(* CODESYS project CtaAppSperrAntrieb_2.0.0.0.library
   Description: Sperr- Antriebs Library der CTA
   Version: 2.0.0.0
   Title: CtaAppSperrAntrieb
   Author: SIS
   DocFormat: reStructuredText
   Placeholder: CtaAppSperrAntrieb
   LanguageModelAttribute: qualified-access-only
   CompiledLibraryCompatibilityVersion: CODESYS V3.5 SP16 Patch 3
   Company: CTA
   DefaultNamespace: CtaAppSperrAntrieb

Project tree, tasks and I/O mapping:
  libraries: Standard, 3.5.18.0 (System); CtaAppBasic, 1.0.0.0 (CTA); CtaAppBmk, 2.0.0.0 (CTA); CtaAppReport, 2.0.0.0 (CTA); CtaSysConfig, 2.0.0.0 (CTA); VisuSymbols, 4.5.0.0 (System); VisuDialogs, 3.5.16.20 (System); CtaSysMotor, 1.0.0.0 (CTA); CtaVisHelp, 1.0.0.0 (CTA); CtaVisSymbols, 2.0.0.0 (CTA); CtaSysIO, 2.0.0.0 (CTA); CtaAppInfluxLog, 1.0.0.1 (CTA); CtaAppModbusSpezifikation, 1.0.0.1 (CTA); CtaVisApps, 1.0.0.0 (CTA); CtaVisUser, 1.0.0.0 (CTA)
  40 Visualizations/
    ICON/
      SperrAntrieb_RIGHT/
        Motor_Right/
          Above/
            visualisation SperrAntrieb_MR_Flap_Txt_R_Above
            visualisation SperrAntrieb_MR_Flap_RA_CheckQuerry
            visualisation SperrAntrieb_MR_Flap_RA_CheckEnabled
          Below/
            visualisation SperrAntrieb_MR_Flap_Txt_R_Below
            visualisation SperrAntrieb_MR_Flap_RB_CheckQuerry
            visualisation SperrAntrieb_MR_Flap_RB_CheckEnabled
        Motor_Above/
          visualisation SperrAntrieb_MA_Flap_RA_CheckEnabled
          visualisation SperrAntrieb_MA_Flap_RA_CheckQuerry
          visualisation SperrAntrieb_MA_Flap_Txt_R_Above
        Motor_Below/
          visualisation SperrAntrieb_MB_Flap_RB_CheckEnabled
          visualisation SperrAntrieb_MB_Flap_RB_CheckQuerry
          visualisation SperrAntrieb_MB_Flap_Right_Txt_R_Below
        Motor_Left/
          Above/
            visualisation SperrAntrieb_ML_Flap_Txt_R_Above
            visualisation SperrAntrieb_ML_Flap_RA_CheckQuerry
            visualisation SperrAntrieb_ML_Flap_RA_CheckEnabled
          Below/
            visualisation SperrAntrieb_ML_Flap_Txt_R_Below
            visualisation SperrAntrieb_ML_Flap_RB_CheckQuerry
            visualisation SperrAntrieb_ML_Flap_RB_CheckEnabled
      SperrAntrieb_BASE/
        Ventile/
          Klappe/
            Motor_Left/
              visualisation ML_Klappe_ZU
              visualisation ML_Klappe_AUF
            Motor_Below/
              visualisation MB_Klappe_ZU
              visualisation MB_Klappe_AUF
            Motor_Above/
              visualisation MA_Klappe_ZU
              visualisation MA_Klappe_AUF
            Motor_Right/
              visualisation MR_Klappe_ZU
              visualisation MR_Klappe_AUF
        Icons/
          visualisation Motor
          Motor_Left/
            visualisation Icon_ML_Klappe
          Motor_Right/
            visualisation Icon_MR_Klappe
          Motor_Below/
            visualisation Icon_MB_Klappe
          Motor_Above/
            visualisation Icon_MA_Klappe
        Value/
          visualisation ValueUpDwn
          visualisation ValueDwnUp
      SperrAntrieb_LEFT/
        Motor_LEFT/
          Above/
            visualisation SperrAntrieb_ML_Flap_Txt_L_Above
            visualisation SperrAntrieb_ML_Flap_LA_CheckQuerry
            visualisation SperrAntrieb_ML_Flap_LA_CheckEnabled
          Below/
            visualisation SperrAntrieb_ML_Flap_Txt_L_Below
            visualisation SperrAntrieb_ML_Flap_LB_CheckQuerry
            visualisation SperrAntrieb_ML_Flap_LB_CheckEnabled
        Motor_Above/
          visualisation SperrAntrieb_MA_Flap_LA_CheckQuerry
          visualisation SperrAntrieb_MA_Flap_Txt_L_Above
          visualisation SperrAntrieb_MA_Flap_LA_CheckEnabled
        Motor_Below/
          visualisation SperrAntrieb_MB_Flap_LB_CheckEnabled
          visualisation SperrAntrieb_MB_Flap_LB_CheckQuerry
          visualisation SperrAntrieb_MB_Flap_Txt_L_Below
        Motor_Right/
          Above/
            visualisation SperrAntrieb_MR_Flap_Txt_L_Above
            visualisation SperrAntrieb_MR_Flap_LA_CheckQuerry
            visualisation SperrAntrieb_MR_Flap_LA_CheckEnabled
          Below/
            visualisation SperrAntrieb_MR_Flap_Txt_L_Below
            visualisation SperrAntrieb_MR_Flap_LB_CheckQuerry
            visualisation SperrAntrieb_MR_Flap_LB_CheckEnabled
    POPUP/
      visualisation SperrAntrieb_POPUP
      PARAMETER/
        visualisation SperrAntrieb_PARAMETER
        visualisation SperrAntrieb_ParameterListe
        SperrAntrieb_ParameterBase/
          visualisation SperrAntrieb_ParameterBase0
          visualisation SperrAntrieb_ParameterBase
        SperrAntrieb_Fuse/
          visualisation SperrAntrieb_ParameterFuses0
          visualisation SperrAntrieb_ParameterFuses
        SperrAntrieb_IO/
          visualisation SperrAntrieb_ParameterIO0
          visualisation SperrAntrieb_ParameterIO1
          visualisation SperrAntrieb_ParameterIO
          visualisation SperrAntrieb_ParameterIO2
          visualisation SperrAntrieb_ParameterIO3
          visualisation SperrAntrieb_ParameterIO4
        SperrAntrieb_InfluxDb/
          visualisation SperrAntrieb_ParameterInfluxDb
          visualisation SperrAntrieb_ParameterInfluxDb0
        visualisation SperrAntrieb_Icon_SperrAntrieb
        visualisation SperrAntrieb_POPUP_IO_ITF
      visualisation SperrAntrieb_PopUpListe
      MANUAL/
        visualisation SperrAntrieb_MANUAL
      OVERVIEW/
        visualisation SperrAntrieb_OVERVIEW
      BUS/
        visualisation SperrAntrieb_BUS
        visualisation SperrAntrieb_BUS_SW0_Detail
        visualisation SperrAntrieb_BUS_CW0_Detail
        visualisation SperrAntrieb_BUS_CS
        visualisation SperrAntrieb_BUS_SW1_Detail
        visualisation SperrAntrieb_BUS_SW2_Detail
      REPORTS/
        visualisation SperrAntrieb_REPORTS
      IO/
        visualisation SperrAntrieb_IO0
        visualisation SperrAntrieb_IO
        visualisation SperrAntrieb_IO1
  30 Program Organization Units/
    function block fbSperrAntrieb [ST]: proHandOn, proAuto, proHandOff, proHandManualClose, proHardWareHandModulAktive, proHandManualOpen, actConfig, proConfigError, proValveIcon, p_scActuatorFuse_fbxEnable, p_scActuatorFuse_fbxInputMb, p_scActuatorFuse_fbxDoesAlarm, p_scBase_fbxEnable, p_scBase_fbxControllMb, p_scBase_fbxInvertiert, p_scBase_fbtSettingTime, p_scFuse_fbxEnable, p_scFuse_fbxInputMb, p_scFuse_fbxDoesAlarm, p_scInSperrAtRevisionSwitch_fbxEnable, p_scInSperrAtRevisionSwitch_fbxInputMb, p_scInSperrAtReady_fbxEnable, p_scInSperrAtReady_fbxInputMb, p_scInSperrAtHand_fbxEnable, p_scInSperrAtHand_fbxInputMb, p_scInSperrAtRükClosed_fbxEnable, p_scInSperrAtRükClosed_fbxInputMb, p_scInSperrAtRükClosed_fbxDoesAlarm, p_scInSperrAtRükClosed_fbtDelayStart, p_scInSperrAtRükClosed_fbtDelayRun, p_scInSperrAtRükClosed_fbiTypeOfAck, p_scInSperrAtRükClosed_fbiMaxErrorRetryAllowed, p_scInSperrAtRükOpen_fbxEnable, p_scInSperrAtRükOpen_fbxInputMb, p_scInSperrAtRükOpen_fbxDoesAlarm, p_scInSperrAtRükOpen_fbtDelayStart, p_scInSperrAtRükOpen_fbtDelayRun, p_scInSperrAtRükOpen_fbiTypeOfAck, p_scInSperrAtRükOpen_fbiMaxErrorRetryAllowed, p_scInSperrAtActualPosition_fbxEnable, p_scInSperrAtActualPosition_fbxInputMb, p_scInSperrAtActualPosition_fbxDoesAlarm, p_scInSperrAtActualPosition_fbrMaxDiff, p_scInSperrAtActualPosition_fbtDelayStart, p_scInSperrAtActualPosition_fbtDelayRun, p_scInSperrAtActualPosition_fbiTypeOfAck, p_scInSperrAtActualPosition_fbiMaxErrorRetryAllowed, p_scManual_fbxAlowManualOn, p_scManual_fbuiManualState, p_scManual_fbuiSchaltBefehl, p_scInfluxDb_fbxEnable, actMbControll, actMbState, proModbusTest, proModbusStateWord, proModbusControllWord, proKlappenStatus, proIsError, proIsWarning, proIsRegulatet, proIsEnabled, actState, proIsHandOnOrOff, proIsReady, proIsOnY, proRevisionSwitchOk, proStateSymbol, proAnzError, proAnzInfo, proAnzWarning, proITF_REPORTMANAGER, proIsInverted, proRükIsClosed, proRükIsOpen, proOn, metDI_RükIsOpen, proGetDI_RükIsOpen, proNotShowDI_RükIsOpen, proIsOpen_ITF, metDI_RükIsClosed, proGetDI_RükIsClosed, proNotShowDI_RükIsClosed, proIsClosed_ITF, metDI_RevisionSwitchOk, proNotShowDI_RevisionSwitchOk, proGetDI_RevisionSwitchOK, proRevisionSwitch_ITF, proGetDI_FuseOK, metDI_FuseOK, proNotShowDI_FuseOk, proFuse_ITF, metDI_ActuatorHand, proNotShowDI_ActuatorHand, proGetDI_ActuatorHand, proHandModul_ITF, metDI_IsReady, proNotShowDI_Ready, proGetDI_IsReady, proActuatorReady_ITF, metDI_ActuatorFuseOk, proNotShowDI_ActuatorFuseOk, proGetDI_ActuatorFuseOk, proActuatorFuse_ITF, proActualPosition_ITF, metAI_ActualPosition, proNotShowAI_ActualPosition, proGetAI_ActualPosition, proOnY_ITF, metAO_OnY, proOnOpen_ITF, metDO_xOnAuf, proOnClose_ITF, metDO_xOnZu, proOnY, actPrioOfControll, actResetOnDisable, proOnAuf, proOnZu, proEn, proEnSymbol, actTrendLog, actReport, proAcknowlege, proAvailable, proLockDown
    function fcGetBigerStringValue [ST]
    Abstracte Bausteine/
    function fcCheckQuerryReturnIcon [ST]
  00000000-0000-0000-0000-000000000000|D:\CoDeSys\LibrariesV3\trunk\Intern\CAA\CAA Template\3.4.0.0 draft\Placeholder.xml
  00000000-0000-0000-0000-000000000000|D:\CoDeSys\LibrariesV3\trunk\Intern\CAA\CAA Template\3.2.0.3 draft\Prefix.pdf
  00000000-0000-0000-0000-000000000000|D:\CoDeSys\LibrariesV3\trunk\Intern\CAA\CAA Template\3.5.2.0 draft\Placeholder.xml
  20 Structs/
    data type scParameter
    STATE/
      data type scInSperrAtReady
      data type scInSperrAtRevisionSwitch
      data type scInSperrAtActualPosition
      data type scInSperrAtHand
      data type scInSperrAtRükOpen
      data type scInSperrAtRükClosed
    BASE/
      data type scBase
    FUSE/
      data type scFuse
      data type scActuatorFuse
    InfluxDb/
      data type scInfluxDb
    MANUAL/
      data type scManual
    data type enKlappenStatus
  50 Images/
  10 Documenation/
    global variables VersionHistory
    global variables readMe
  21 Interface/
    interface ITF_SPERRANTRIEB: proAuto, proHandOff, proHandOn, proIsRegulatet, proIsError, proIsWarning, proIsEnabled, proIsHandOnOrOff, proIsReady, proHardWareHandModulAktive, proRevisionSwitchOk, proHandManualClose, proEn, proRükIsOpen, proRükIsClosed, proStateSymbol, proEnSymbol, proOnZu, proIsOnY, proOnAuf, proOnY, proGetDI_RükIsOpen, proNotShowDI_RükIsOpen, proIsOpen_ITF, proGetDI_ActuatorHand, proNotShowDI_ActuatorHand, proHandModul_ITF, proGetDI_ActuatorFuseOk, proNotShowDI_ActuatorFuseOk, proActuatorFuse_ITF, proGetDI_IsReady, proNotShowDI_Ready, proActuatorReady_ITF, proGetDI_FuseOK, proNotShowDI_FuseOk, proFuse_ITF, proGetDI_RevisionSwitchOK, proNotShowDI_RevisionSwitchOk, proRevisionSwitch_ITF, proNotShowAI_ActualPosition, proGetAI_ActualPosition, proActualPosition_ITF, proGetDI_RükIsClosed, proNotShowDI_RükIsClosed, proIsClosed_ITF, proOnY_ITF, proOnOpen_ITF, proOnClose_ITF, proAnzWarning, proITF_REPORTMANAGER, proAnzInfo, proAnzError, proModbusTest, proModbusStateWord, proModbusControllWord, proConfigError, p_scBase_fbxEnable, p_scBase_fbxControllMb, p_scBase_fbxInvertiert, p_scBase_fbtSettingTime, p_scFuse_fbxEnable, p_scFuse_fbxInputMb, p_scFuse_fbxDoesAlarm, p_scActuatorFuse_fbxEnable, p_scActuatorFuse_fbxInputMb, p_scActuatorFuse_fbxDoesAlarm, p_scInSperrAtRevisionSwitch_fbxEnable, p_scInSperrAtRevisionSwitch_fbxInputMb, p_scInSperrAtReady_fbxEnable, p_scInSperrAtReady_fbxInputMb, p_scInSperrAtHand_fbxEnable, p_scInSperrAtHand_fbxInputMb, p_scInSperrAtRükClosed_fbxEnable, p_scInSperrAtRükClosed_fbxInputMb, p_scInSperrAtRükClosed_fbxDoesAlarm, p_scInSperrAtRükClosed_fbtDelayStart, p_scInSperrAtRükClosed_fbtDelayRun, p_scInSperrAtRükClosed_fbiTypeOfAck, p_scInSperrAtRükClosed_fbiMaxErrorRetryAllowed, p_scInSperrAtRükOpen_fbxEnable, p_scInSperrAtRükOpen_fbxInputMb, p_scInSperrAtRükOpen_fbxDoesAlarm, p_scInSperrAtRükOpen_fbtDelayStart, p_scInSperrAtRükOpen_fbtDelayRun, p_scInSperrAtRükOpen_fbiTypeOfAck, p_scInSperrAtRükOpen_fbiMaxErrorRetryAllowed, p_scInSperrAtActualPosition_fbxEnable, p_scInSperrAtActualPosition_fbxInputMb, p_scInSperrAtActualPosition_fbxDoesAlarm, p_scInSperrAtActualPosition_fbrMaxDiff, p_scInSperrAtActualPosition_fbtDelayStart, p_scInSperrAtActualPosition_fbtDelayRun, p_scInSperrAtActualPosition_fbiTypeOfAck, p_scInSperrAtActualPosition_fbiMaxErrorRetryAllowed, p_scInfluxDb_fbxEnable, p_scManual_fbxAlowManualOn, p_scManual_fbuiManualState, p_scManual_fbuiSchaltBefehl, proHandManualOpen, proIsInverted, proKlappenStatus, proValveIcon, proAcknowlege, proAvailable, proLockDown, proOn
  11 Library Parameter/
    global variables Parameter
  12 Konstanten/
    global variables GlobalKonstant
  60 Textlisten/
    text list GlobalTextList
    text list Error
    text list Info
    text list Warnung
    text list KlappenStatus
  13 Globale Variablen/
  5ce3da45-db07-42e7-a21c-a00fff4ed8f6|C:\Users\sis\Downloads\dip-switch.svg
  5ce3da45-db07-42e7-a21c-a00fff4ed8f6|C:\Users\sis\Downloads\lightning-bolt-circle.svg
  5ce3da45-db07-42e7-a21c-a00fff4ed8f6|C:\Users\sis\Downloads\sine-wave.svg
  5ce3da45-db07-42e7-a21c-a00fff4ed8f6|C:\Users\sis\Downloads\eye.svg
  5ce3da45-db07-42e7-a21c-a00fff4ed8f6|C:\Users\sis\Downloads\lan.svg
*)

// 20 Structs/scParameter
{attribute 'pack_mode' := '1'} 
TYPE scParameter :
    STRUCT
        scBase              		:   scBase;
        scFuse              		:   scFuse;
        scActuatorFuse         		:   scActuatorFuse;
        scInSperrAtRevisionSwitch	:   scInSperrAtRevisionSwitch;
        scInSperrAtReady         	:   scInSperrAtReady; 
        scInSperrAtActualPosition   :   scInSperrAtActualPosition;
		scInSperrAtRükOpen			:	scInSperrAtRükOpen;
		scInSperrAtRükClosed		:	scInSperrAtRükClosed;
        scManual            		:   scManual;
        scInfluxDb          		:   scInfluxDb;
        scInSperrAtHand          	:   scInSperrAtHand;
    END_STRUCT
END_TYPE

// 20 Structs/STATE/scInSperrAtReady
{attribute 'pack_mode' := '1'} 
TYPE scInSperrAtReady :
    STRUCT
        fbxEnable                    : CtaSysConfig.fbBOOL;
        fbxInputMb                   : CtaSysConfig.fbBOOL;          
    END_STRUCT
END_TYPE

// 20 Structs/STATE/scInSperrAtRevisionSwitch
{attribute 'pack_mode' := '1'} 
TYPE scInSperrAtRevisionSwitch :
    STRUCT
        fbxEnable                   : CtaSysConfig.fbBOOL;
        fbxInputMb                  : CtaSysConfig.fbBOOL;           
    END_STRUCT
END_TYPE

// 20 Structs/STATE/scInSperrAtActualPosition
{attribute 'pack_mode' := '1'} 
TYPE scInSperrAtActualPosition :
    STRUCT
        fbxEnable                    : CtaSysConfig.fbBOOL;
        fbxInputMb                   : CtaSysConfig.fbBOOL;   
        fbxDoesAlarm                 : CtaSysConfig.fbBOOL;  
        fbrMaxDiff                   : CtaSysConfig.fbREAL;
        fbtDelayStart                : CtaSysConfig.fbTIME;
        fbtDelayRun                  : CtaSysConfig.fbTIME;
		fbiTypeOfAck               	 : CtaSysConfig.fbINT;   
        fbiMaxErrorRetryAllowed      : CtaSysConfig.fbINT;         
    END_STRUCT
END_TYPE

// 20 Structs/STATE/scInSperrAtHand
{attribute 'pack_mode' := '1'} 
TYPE scInSperrAtHand :
    STRUCT
        fbxEnable                   : CtaSysConfig.fbBOOL;    
        fbxInputMb                  : CtaSysConfig.fbBOOL; 
    END_STRUCT
END_TYPE

// 20 Structs/BASE/scBase
{attribute 'pack_mode' := '1'} 
TYPE scBase :
    STRUCT
        fbxEnable       		:   CtaSysConfig.fbBOOL;
		fbxControllMb   		:   CtaSysConfig.fbBOOL;
		fbxInvertiert			:	CtaSysConfig.fbBOOL;
		fbtSettingTime			:	CtaSysConfig.fbTIME;		
    END_STRUCT
END_TYPE

// 20 Structs/FUSE/scFuse
{attribute 'pack_mode' := '1'} 
TYPE scFuse :
    STRUCT
        fbxEnable               : CtaSysConfig.fbBOOL;
        fbxInputMb              : CtaSysConfig.fbBOOL;
        fbxDoesAlarm            : CtaSysConfig.fbBOOL;
    END_STRUCT
END_TYPE

// 20 Structs/FUSE/scActuatorFuse
{attribute 'pack_mode' := '1'} 
TYPE scActuatorFuse :
    STRUCT
        fbxEnable             : CtaSysConfig.fbBOOL;
        fbxInputMb            : CtaSysConfig.fbBOOL;
        fbxDoesAlarm          : CtaSysConfig.fbBOOL;      
    END_STRUCT
END_TYPE

// 20 Structs/InfluxDb/scInfluxDb
{attribute 'pack_mode' := '1'} 
TYPE scInfluxDb :
    STRUCT
        fbxEnable       :   CtaSysConfig.fbBOOL;
    END_STRUCT
END_TYPE

// 20 Structs/MANUAL/scManual
{attribute 'pack_mode' := '1'} 
TYPE scManual :
    STRUCT
        fbxAlowManualOn         : CtaSysConfig.fbBOOL;    
        fbuiManualState         : CtaSysConfig.fbUINT;          // 0 = Auto, 1 = Manual Off, 2 = Manual On
        fbuiSchaltBefehl		: CtaSysConfig.fbUINT;			// 0 = Idle, 1 = Schliessen, 2 = Öffnen 
    END_STRUCT
END_TYPE

// 20 Structs/STATE/scInSperrAtRükOpen
TYPE scInSperrAtRükOpen :
	STRUCT
		fbxEnable                    : CtaSysConfig.fbBOOL;
		fbxInputMb                   : CtaSysConfig.fbBOOL;   
		fbxDoesAlarm                 : CtaSysConfig.fbBOOL;  
		fbtDelayStart                : CtaSysConfig.fbTIME;
		fbtDelayRun                  : CtaSysConfig.fbTIME;
		fbiTypeOfAck               	 : CtaSysConfig.fbINT;   
        fbiMaxErrorRetryAllowed      : CtaSysConfig.fbINT;      
	END_STRUCT
END_TYPE

// 20 Structs/STATE/scInSperrAtRükClosed
TYPE scInSperrAtRükClosed :
	STRUCT
		fbxEnable                    : CtaSysConfig.fbBOOL;
		fbxInputMb                   : CtaSysConfig.fbBOOL;   
		fbxDoesAlarm                 : CtaSysConfig.fbBOOL;  
		fbtDelayStart                : CtaSysConfig.fbTIME;
		fbtDelayRun                  : CtaSysConfig.fbTIME;
		fbiTypeOfAck               	 : CtaSysConfig.fbINT;   
        fbiMaxErrorRetryAllowed      : CtaSysConfig.fbINT;    
	END_STRUCT
END_TYPE

// 20 Structs/enKlappenStatus
{attribute 'qualified_only'}
{attribute 'strict'}
TYPE enKlappenStatus :
(	
	Gesperrt 	:= 0,
	Schliesst	, 
	IstZu		,
	Öffnet		,
	IstOffen	,
	Idle		
);
END_TYPE

// 10 Documenation/VersionHistory
(* 

.. image:: ../../Images/CTA_Logo.jpg
   :align: right
   :width: 15% 

**Vorlage**   


============ =========== =========== ============================================
**Date**     **Version** **Author**  **Change**
------------ ----------- ----------- --------------------------------------------
04.03.2021   0.0.0.0     SIS         Vorlage erstellt

============ =========== =========== ============================================


*)
VAR_GLOBAL
    stInfo : STRING:= '0.0.0.0, Vorlage, CTA';
END_VAR

// 10 Documenation/readMe
(*

**ReadMe**
 
|	**Empfehlung**
|
|	Biblitothek CtaAppSperrAntrieb zur Ansteuerung von Sperrantrieben
|	Instanzieren Sie den CtaAppSperrAntrieb.fbSperrAntrieb in ihrem Funktionsbaustein oder POU beispielsweise als fbSperAX. (X = Nr.) 
|	Deklarieren Sie die Struktur Variable welche als Parameter und zur ansteuerung dienen wie im Code beispiel.
|  
| *Beispiel* 

+-----------------------+---------------------------------------------------------------------------------------------------------------------------------------------------------------------------------------------------------------------------------------------------------------------------------------------------------------------------------------------------------------------------------------------------------------------------------------+
| Beschreibung          |  Code                                                                                                                                                                                                                                                                                                                                                                                                                                 |
+=======================+=======================================================================================================================================================================================================================================================================================================================================================================================================================================+
| Pou oder SmFb         | .. code-block:: codesys                                                                                                                                                                                                                                                                                                                                                                                                               |
|                       |                                                                                                                                                                                                                                                                                                                                                                                                                                       |
|                       |	// Deklaration als VAR im POU oder dem selbsterstellten Funktionsbaustein                                                                                                                                                                                                                                                                                                                                                        	|
|                       |   VAR   																																																				 																																																				|
|						|	    (*Sperrantrieb 1*)																																																		 																																																		|
|						|		fbSperA1			: CtaAppSperrAntrieb.fbSperrAntrieb;                                                                                                                                                                                                                                                                                                                                                               			|
|                       | 		(*Sperrantrieb 2*)																																																		 																																																		|
|			 			|		fbSperA2			: CtaAppSperrAntrieb.fbSperrAntrieb;																																												 																																														|
|			 			|	END_VAR                                                                                                                                                                                                                                                                                                                                                                                                                          	|
+-----------------------+---------------------------------------------------------------------------------------------------------------------------------------------------------------------------------------------------------------------------------------------------------------------------------------------------------------------------------------------------------------------------------------------------------------------------------------+
| Code für Init         | .. code-block:: codesys                                                                                                                                                                                                                                                                                                                                                                                                               |
|                       |   																																																					 																																																				|
|			 			|	// Kopieren des nachfolgenden Codes in eine Action zur Initialisierung der Parameter. Zum Beispiel actConfig.																																																				 																										|
|                       |	{region "Parameter Sperrantrieb1"}                                                                                                                                                                                                                                                                                                                                                                                                 	|
|			 			|		(*Basis*)                                                                                                                                                                                                                                                                                                                                                                                                                       |
|						|		fbSperA1.scParameter.scBase.fbxEnable                					(_WertInit :=  TRUE																		 );		//P1 Ein- Ausschalten des Sperrantriebs                                                                                                                                                                                                           		|
|						|		fbSperA1.scParameter.scBase.fbxControllMb 								(_WertInit :=  TRUE																		 );     //P2 Ansteuerung oder Signalauswertung über Modbus                                                                                                                                                                                            			|
|						|		fbSperA1.scParameter.scBase.fbxInvertiert								(_WertInit := FALSE																		 );     //P3 Stellantrieb Invertierung                                                                                                                                                                                                                  		|
|						|		fbSperA1.scParameter.scBase.fbtSettingTime								(_WertInit := T#00S									, _minInit :=      , _maxInit:= 	 );     //P4 Stellzeit der Klappe                                                                                                                                                                                                                            	|
|						|		(*Fuse Parameter*)                                                                                                                                                                                                                                                                                                                                                                                           					|
|						|		fbSperA1.scParameter.scFuse.fbxEnable   								(_WertInit := FALSE																		 );     //P5 Sicherung ist vorhanden / nicht vorhanden                                                                                                                                          																|
|						|		fbSperA1.scParameter.scFuse.fbxInputMb  								(_WertInit := FALSE																		 );     //P6 Ansteuerung oder Signalauswertung über Modbus                                                                                                                                                                                                      |
|						|		fbSperA1.scParameter.scFuse.fbxDoesAlarm								(_WertInit := FALSE																		 );     //P7 Abfallendes Signal löst Fehler aus                                                                                                                                                                                                   				|
|						|		(*Stellantrieb Fuse Parameter*)       																																																																																															|
|						|		fbSperA1.scParameter.scActuatorFuse.fbxEnable                   		(_WertInit := FALSE																		 );     //P8 Leistungsschutzschalter ist vorhanden / nicht vorhanden                                                                                                                                                                                            |
|						|		fbSperA1.scParameter.scActuatorFuse.fbxInputMb   						(_WertInit := FALSE																		 );     //P9 Ansteuerung oder Signalauswertung über Modbus                                                                                                                                                                                                      |
|						|		fbSperA1.scParameter.scActuatorFuse.fbxDoesAlarm 						(_WertInit := FALSE																		 );     //P10 Abfallendes Signal löst Fehler aus                                                                                                                                                                                                                |
|						|		(*Revision Switch Parameter*)                                 		                                                                                                                                                                                                                                                                                                                                                        	|
|						|		fbSperA1.scParameter.scInSperrAtRevisionSwitch.fbxEnable  				(_WertInit := FALSE																		 );     //P11 Revisionschalter ist vorhanden / nicht vorhanden                                                                                                                                                                         							|
|						|		fbSperA1.scParameter.scInSperrAtRevisionSwitch.fbxInputMb 				(_WertInit := FALSE																		 );     //P12 Ansteuerung oder Signalauswertung über Modbus                                                                                                                                                                                                     |
|						|		(*Ready Input Parameter*)                                                                                                                                                                                                                                                                                                                                                                                                     	|
|						|		fbSperA1.scParameter.scInSperrAtReady.fbxEnable  						(_WertInit := FALSE																		 );     //P13 Readysignal ist vorhanden / nicht vorhanden                                                                                                                                                                                                       |
|						|		fbSperA1.scParameter.scInSperrAtReady.fbxInputMb 						(_WertInit := FALSE																		 );     //P14 Ansteuerung oder Signalauswertung über Modbus                                                                                                                                                                                                     |
|						|		(*Stellantrieb Input Hand*)         							                                                                                                                                                                                                                                                                                                                                                                |
|						|		fbSperA1.scParameter.scInSperrAtHand.fbxEnable 							(_WertInit := FALSE																		 );     //P15 Handmodul ist vorhanden / nicht vorhanden                                                                                                                                                                                                         |
|						|		fbSperA1.scParameter.scInSperrAtHand.fbxInputMb							(_WertInit := FALSE																		 );     //P16 Ansteuerung oder Signalauswertung über Modbus                                                                                                                                                                                                     |
|						|		(*Is closed Input Parameter*)                     	        	                                                                                                                                                                                                                                                                                                                                                            	|
|						|		fbSperA1.scParameter.scInSperrAtRükClosed.fbxEnable		 				(_WertInit := FALSE																		 );     //P17 Rückmeldung ZU ist vorhanden / nicht vorhanden                                                                                                                                                                                                    |
|						|		fbSperA1.scParameter.scInSperrAtRükClosed.fbxInputMb      				(_WertInit := FALSE																		 );     //P18 Ansteuerung oder Signalauswertung über Modbus                                                                                                                                                                                                     |
|						|		fbSperA1.scParameter.scInSperrAtRükClosed.fbxDoesAlarm    				(_WertInit := FALSE																		 );     //P19 Fehlendes oder abfallendes Signal löst Fehler aus                                                                                                                                                             									|
|						|		fbSperA1.scParameter.scInSperrAtRükClosed.fbtDelayStart   				(_WertInit := T#00S									, _minInit :=      , _maxInit:= 	 );     //P20 Verzögerung der Fehlerausgabe nach Start                                                                                                                                                                                                          |
|						|		fbSperA1.scParameter.scInSperrAtRükClosed.fbtDelayRun     				(_WertInit := T#00S									, _minInit :=      , _maxInit:= 	 );     //P21 Verzögerung der Fehlerausgabe während Betrieb                                                                                                                                                                                                     |
|						|		fbSperA1.scParameter.scInSperrAtRükClosed.fbiTypeOfAck					(_WertInit :=     0									, _minInit :=     0, _maxInit:=     2);     //P22 Art der Quittierung des Fehlers (auto, quittierned, quittiernd bis n meldung)                                                                                                                                                                     |
|						|		fbSperA1.scParameter.scInSperrAtRükClosed.fbiMaxErrorRetryAllowed		(_WertInit :=     3									, _minInit :=     0, _maxInit:= 	5);     //P23 Maximale Anzahl Wiederholungen bis zu Sperrung der Anlage                                                                                                                                                                           				|
|						|		(*Is open Input Parameter*)                       			                                                                                                                                                                                                                                                                                                                                                                	|
|						|		fbSperA1.scParameter.scInSperrAtRükOpen.fbxEnable		 				(_WertInit := FALSE																		 );     //P24 Rückmeldung OFFEN ist vorhanden / nicht vorhanden                                                                                                                                                                                                 |
|						|		fbSperA1.scParameter.scInSperrAtRükOpen.fbxInputMb        				(_WertInit := FALSE																		 );     //P25 Ansteuerung oder Signalauswertung über Modbus                                                                                                                                                                                                    	|
|						|		fbSperA1.scParameter.scInSperrAtRükOpen.fbxDoesAlarm      		    	(_WertInit := FALSE																		 );     //P26 Fehlendes oder abfallendes Signal löst Fehler aus                                                                                                                                                                                                	|
|						|		fbSperA1.scParameter.scInSperrAtRükOpen.fbtDelayStart     				(_WertInit := T#00S									, _minInit :=      , _maxInit:= 	 );     //P27 Verzögerung der Fehlerausgabe nach Start                                                                                                                                                                                                         	|
|						|		fbSperA1.scParameter.scInSperrAtRükOpen.fbtDelayRun       				(_WertInit := T#00S									, _minInit :=      , _maxInit:= 	 );     //P28 Verzögerung der Fehlerausgabe während Betrieb                                                                                                                                                                                                    	|
|						|		fbSperA1.scParameter.scInSperrAtRükOpen.fbiTypeOfAck					(_WertInit :=     0									, _minInit :=     0, _maxInit:=     2);     //P29 Art der Quittierung des Fehlers  (auto, quittierned, quittiernd bis n meldung)                                                                                                                                                                    |
|						|		fbSperA1.scParameter.scInSperrAtRükOpen.fbiMaxErrorRetryAllowed			(_WertInit :=     3									, _minInit :=     0, _maxInit:= 	5);     //P30 Maximale Anzahl Wiederholungen bis zu Sperrung der Anlage                                                                                                                                                                                      	|
|						|		(*Actual value Input Parameter*)                          	                                                                                                                                                                                                                                                                                                                                                                	|
|						|		fbSperA1.scParameter.scInSperrAtActualPosition.fbxEnable     			(_WertInit := FALSE																		 );     //P31 Rückmeldung des Istwerts ist vorhanden / nicht vorhanden                                                                                                                                                                                          |
|						|		fbSperA1.scParameter.scInSperrAtActualPosition.fbxInputMb    			(_WertInit := FALSE																		 );     //P32 Ansteuerung oder Signalauswertung über Modbus                                                                                                                                                                                                   	|
|						|		fbSperA1.scParameter.scInSperrAtActualPosition.fbxDoesAlarm  			(_WertInit := FALSE																		 );     //P33 Unter oder überschreitung der Maximal erlaubten Differenz löst Fehler aus                                                                                                                                                            				|
|						|		fbSperA1.scParameter.scInSperrAtActualPosition.fbrMaxDiff    			(_WertInit :=   0.0									, _minInit :=      , _maxInit:=      );     //P34 Maximal erlaubte Differenz des Stell- zum Istwert                                                                                                                                                   	 											|
|						|		fbSperA1.scParameter.scInSperrAtActualPosition.fbtDelayStart 			(_WertInit := T#00S									, _minInit :=      , _maxInit:= 	 );     //P35 Verzögerung der Fehlerausgabe nach Start                                                                                                                                        					  												|
|						|		fbSperA1.scParameter.scInSperrAtActualPosition.fbtDelayRun   			(_WertInit := T#00S									, _minInit :=      , _maxInit:= 	 );     //P36 Verzögerung der Fehlerausgabe während Betrieb                                                                                                                                               														|
|						|		fbSperA1.scParameter.scInSperrAtActualPosition.fbiTypeOfAck				(_WertInit :=     0									, _minInit :=     0, _maxInit:=     2);     //P37 Art der Quittierung des Fehlers (auto, quittierned, quittiernd bis n meldung)                                                                                                       																|
|						|		fbSperA1.scParameter.scInSperrAtActualPosition.fbiMaxErrorRetryAllowed	(_WertInit :=     3									, _minInit :=     0, _maxInit:= 	5);     //P38 Maximale Anzahl Wiederholungen bis zu Sperrung der Anlage                                                                                                                                   														|
|						|		(*InfluxDb*)                                                                                                                                                                                                                                                                                                                                                                                                                  	|
|						|		fbSperA1.scParameter.scInfluxDb.fbxEnable                               (_WertInit := FALSE																		 );     //P39 Aktivierung / Deaktivierung der Trenddaten                                                                                                                                                                                                     	|
|						|		(*Manual Parameter*)                                                                                                                                                                                                                                                                                                                                                                                                          	|
|						|		fbSperA1.scParameter.scManual.fbxAlowManualOn                           (_WertInit := FALSE																		 );     //P40 Handansteuerung zulassen / nicht zulassen                                                                                                                                                                                                       	|
|						|		fbSperA1.scParameter.scManual.fbuiManualState                           (_WertInit :=     0									, _minInit :=     0, _maxInit:=     2);     //P41 Ansteuerungsmodus der Klappe (auto, manuell, gesperrt)                                                                                                                                                                             				|
|						|		fbSperA1.scParameter.scManual.fbuiSchaltBefehl                          (_WertInit :=     1									, _minInit :=     0, _maxInit:=     2);     //P42 Schaltbefehl der Klappen (idle, schliessen, öffnen)                                                                                                                                                                                            	|
|						|	{endregion} 	                                                                                                                                                                                                                                                                     																																				|
+-----------------------+---------------------------------------------------------------------------------------------------------------------------------------------------------------------------------------------------------------------------------------------------------------------------------------------------------------------------------------------------------------------------------------------------------------------------------------+
*)                                                                                                                                                                                                                                                                                                                                                                                                                                                               
VAR_GLOBAL
	xReadMeDone              :   BOOL; 
END_VAR

// 11 Library Parameter/Parameter
{attribute 'qualified_only'}
VAR_GLOBAL CONSTANT
    iMaxSperrAntrieb :   INT   := 60;         // Maximale Anzahl verwendeter AT-Bausteine    
END_VAR

// 12 Konstanten/GlobalKonstant
{attribute 'qualified_only'}
VAR_GLOBAL CONSTANT 	
	stReportTextListError   : CtaAppReport.stReportTextList := 'CtaAppSperrAntrieb.Error';
	stReportTextListWarning : CtaAppReport.stReportTextList := 'CtaAppSperrAntrieb.Warnung';
	stReportTextListInfo    : CtaAppReport.stReportTextList := 'CtaAppSperrAntrieb.Info';	
    uiMaxParameter          : UINT := 42;
END_VAR

// 30 Program Organization Units/fbSperrAntrieb
FUNCTION_BLOCK fbSperrAntrieb EXTENDS CtaAppBmk.fbBMK IMPLEMENTS ITF_SPERRANTRIEB 
VAR_INPUT
    xRelease                    	:   BOOL;	
END_VAR                         
VAR_OUTPUT                      
    (* Commmands *)	
	xOnAuf							:	BOOL;	
	xOnZu							:	BOOL;	
    rOnY                        	:   REAL; 	// Stellantrieb Position
	
	(* Status Outputs *)
	xIsOpen							:	BOOL;
	xIsClose						:	BOOL;
END_VAR                 
VAR 
	uiValveIcon						:	UINT;                    
    (* State Intern *)      	
    scEWI                       	:   CtaAppReport.scReportNr;            
    xIsWarning                  	:   BOOL;
    _xIsWarning                 	:   BOOL;	
    xIsError                    	:   BOOL;
    _xIsError                   	:   BOOL;	
    xIsRegulatet                	:   BOOL;	
    xIsEnabled                  	:   BOOL;
    xIsHand                     	:   BOOL;
    xIsHandOn                   	:   BOOL;
    xIsHandOff                  	:   BOOL;
    xIsAuto                     	:   BOOL;
	xIsInverted						:	BOOL;   
    xConfigError                	:   BOOL;	
	xShouldClose					:	BOOL;
	xShouldOpen						:	BOOL;
	(* ITF OUT*)
	ITF_xOnAuf						:	CtaSysIO.ITF_IO;	
	ITF_xOnZu						:	CtaSysIO.ITF_IO;
	ITF_rOnY						:	CtaSysIO.ITF_IO;		
    (* Inputs *)
	(* Aktuelle Position *)
	rActualPosition					:	REAL;	
	rInActualPosition				:	REAL;
	rInActualPositionMb				:	REAL;
	ITF_ActualPosition				:	CtaSysIO.ITF_IO;
	(* Rückmeldung offen *)
	xRückIsOpen						:	BOOL;	
	xInRükIsOpen					:	BOOL;
	xInRükIsOpenMb					:	BOOL;
	ITF_RükIsOpen					:	CtaSysIO.ITF_IO;
	(* Rückmeldung zu*)
	xRückIsClosed					:	BOOL;
	xInRükIsClosed					:	BOOL;
	xInRükIsClosedMb				:	BOOL;
	ITF_RükIsClosed					:	CtaSysIO.ITF_IO;
	(* Generelle Sicherung *)
    xFuseOk                     	:   BOOL;
    xInFuseOk                   	:   BOOL;
    xInFuseOkMb                 	:   BOOL;
	ITF_FuseOk 						:	CtaSysIO.ITF_IO; 
 	(* Stellantriebs sicherung *)
    xActuatorFuseOk                	:   BOOL;    
    xInActuatorFuseOk              	:   BOOL;
    xInActuatorFuseOkMb            	:   BOOL;
	ITF_ActuatorFuseOk				:	CtaSysIO.ITF_IO;
	(* Ready signal *)
    xActuatorIsReady               	:   BOOL;
    xInActuatorIsReady             	:   BOOL;
    xInActuatorIsReadyMb           	:   BOOL;
	ITF_ActuatorIsReady				:	CtaSysIO.ITF_IO;
	(* Revisionsschalter *)
    xActuatorRevisionSwitchOn      	:   BOOL;
    xInActuatorRevisionSwitchOn    	:   BOOL;   
    xInActuatorRevisionSwitchOnMb   :   BOOL;
	ITF_RevisionSwitchOk			:	CtaSysIO.ITF_IO;		
	xActuatorRevisionSwitchOff		:	BOOL;
 	(* Hand Ansteuerung*)
    xActuatorHand                  	:   BOOL;
    xInActuatorHand                	:   BOOL;
    xInActuatorHandMb              	:   BOOL;
	ITF_ActuatorHand				:	CtaSysIO.ITF_IO;  
    (* Freigabe Sperrantrieb *)
    xReleaseFromModBus          	:   BOOL;
    xReleaseControllPrio        	:   BOOL;
     
    (* Modbus *)
    xModbusTest                 	:   BOOL;
    ayMbControllWord            	:   ARRAY[0..3] OF WORD;
    ayMbStateWord               	:   ARRAY[0..3] OF WORD;	
    (* Parameter *)	
    fbConfigFile					:   CtaSysConfig.fbConfigFile;
    scParameter                 	:   scParameter;	
    (* Reports *)	
    fbReportManager			    	:   CtaAppReport.fbReportManager;      
    difor					    	:	DINT;                                                                    
    ayErrorReporter					:	ARRAY[1..6] OF CtaAppReport.fbReporter;
	ayWarningReporter				:	ARRAY[1..4] OF CtaAppReport.fbReporter;
	(*Melder*)
	xErrorDiffAI					:	BOOL;	(*Differenz von Stellwert zu Istwert*)
	xErrorOpenDI					:	BOOL;	(*Keine rückmeldung von Stellventil beim Öffnen*)
	xErrorCloseDI					:	BOOL;	(*Keine Rückmeldung von Stellventil beim Schlissen*)
	(* Trendlogs *)
	fbTrendxOnZu					:	CtaAppInfluxLog.FB_LOG_NODE_BOOL;
	fbTrendxRückIsClosed			:	CtaAppInfluxLog.FB_LOG_NODE_BOOL;
	fbTrendxOnAuf					:	CtaAppInfluxLog.FB_LOG_NODE_BOOL;
	fbTrendxRückIsOpen				:	CtaAppInfluxLog.FB_LOG_NODE_BOOL;
	fbTrendrOnY						:	CtaAppInfluxLog.FB_LOG_NODE_REAL;
	fbTrendrIsOnY					:	CtaAppInfluxLog.FB_LOG_NODE_REAL;
	fbTrendxError					:	CtaAppInfluxLog.FB_LOG_NODE_BOOL;
    (* Collector *)
    diArrayPosition					:   DINT;
	TON_Auf							:	TON;
	TON_Zu							:	TON;
	(*Eingangsüberwachung Digital*)    	
	fbCheckRükOpen					:	CtaSysMotor.fbSafetyInput;
	fbCheckRükClosed				:	CtaSysMotor.fbSafetyInput;		
	(* Eingangsüberwachung Analog*)
	xStellwertOutOk					:	BOOL;
	xNoDiffAI						:	BOOL;
	fbCheckValueAI					:	CtaSysMotor.fbSafetyInput;
END_VAR

(* Config *)
actConfig();

(* Motor Command *)
IF xIsEnabled AND NOT xConfigError THEN
    (* Modbus Controll *)
    actMbControll();
    (* Controll Prio *)
    actPrioOfControll();
	
	(*Klappenansteuerung*)
	(*Manuelle Ansteuerung erlaubt*)
	IF NOT scParameter.scManual.fbxAlowManualOn.proValue THEN
		scParameter.scManual.fbuiManualState.proValue := 0;
	END_IF
		
	(*Automatik*)
	IF scParameter.scManual.fbuiManualState.proValue = 0 THEN
		IF NOT xIsError THEN
			xOnAuf 	:= xReleaseControllPrio XOR scParameter.scBase.fbxInvertiert.proValue;
			xOnZu	:= NOT xReleaseControllPrio XOR scParameter.scBase.fbxInvertiert.proValue;
			rOnY	:= TO_REAL( xReleaseControllPrio XOR scParameter.scBase.fbxInvertiert.proValue) * 100;	
		ELSE
			xOnAuf	:= FALSE XOR scParameter.scBase.fbxInvertiert.proValue;
			xOnZu	:= TRUE	XOR	scParameter.scBase.fbxInvertiert.proValue;
			rOnY	:= TO_REAL(FALSE XOR scParameter.scBase.fbxInvertiert.proValue) * 100;
		END_IF		
		scParameter.scManual.fbuiSchaltBefehl.proValue := 0;
	
	(*Ausgeschalten*)
	ELSIF scParameter.scManual.fbuiManualState.proValue = 1 THEN
		xOnAuf		:= 	FALSE;
		xOnZu		:= 	FALSE;
		rOnY		:= 		0;
		scParameter.scManual.fbuiSchaltBefehl.proValue := 0;
		
	(*Manuelle Ansteuerung*)
	ELSIF scParameter.scManual.fbuiManualState.proValue = 2 THEN
		(*Keine Ansteuerung*)
		IF scParameter.scManual.fbuiSchaltBefehl.proValue = 0 THEN	
			
		
		(* Klappe schliessen *)
		ELSIF scParameter.scManual.fbuiSchaltBefehl.proValue = 1 THEN
			xOnAuf	:= FALSE XOR scParameter.scBase.fbxInvertiert.proValue;
			xOnZu	:= TRUE	XOR scParameter.scBase.fbxInvertiert.proValue;
			rOnY	:= TO_REAL( FALSE XOR scParameter.scBase.fbxInvertiert.proValue) * 100;
		(* Klappe öffnen *)
		ELSIF scParameter.scManual.fbuiSchaltBefehl.proValue = 2 THEN
			xOnAuf	:= TRUE XOR scParameter.scBase.fbxInvertiert.proValue;
			xOnZu	:= FALSE XOR scParameter.scBase.fbxInvertiert.proValue;
			rOnY	:= TO_REAL( TRUE XOR scParameter.scBase.fbxInvertiert.proValue) * 100;			
		END_IF			
	END_IF	
	
	(*Stellwertbegrenzung*)
	IF rOnY >= 100.0 THEN
		rOnY 	:= 100;	
	ELSIF rOnY <= 0.0 THEN
		rOnY	:= 0.0;
	END_IF
	
	(*Timver für Visulaisierungs Darstellung*)
	TON_Zu(	PT := scParameter.scBase.fbtSettingTime.proValue,
			IN := xOnZu);
			
	TON_Auf(PT := scParameter.scBase.fbtSettingTime.proValue,
			IN := xOnAuf);	
	
	(*Eingangsüberwachung Klappenrückmeldung und Signalabfall*)
	(* Digital offen*)
	IF scParameter.scInSperrAtRükOpen.fbxDoesAlarm.proValue > scParameter.scInSperrAtRükOpen.fbxEnable.proValue THEN
		scParameter.scInSperrAtRükOpen.fbxDoesAlarm.proValue := FALSE;
	END_IF
	
	fbCheckRükOpen(		(*Inputs*)
						xSafetyIn 			:= xRückIsOpen ,
						xReferenceIn 		:= xOnAuf,
						(*Parameter*)
						fbxEnSafetyInput 	:= scParameter.scInSperrAtRükOpen.fbxDoesAlarm,
						fbtStartTime 		:= scParameter.scInSperrAtRükOpen.fbtDelayStart,
						fbtRunTime 			:= scParameter.scInSperrAtRükOpen.fbtDelayRun,
						(*Fehler Output*)
						xError				=> xErrorOpenDI );
						
	(*Klappen Rückmeldung offen*)
	IF scParameter.scInSperrAtRükOpen.fbxEnable.proValue THEN
		xIsOpen := xRückIsOpen; 
	ELSE
		xIsOpen := TON_Auf.Q;
	END_IF
	
	(* Digital zu*)
	IF scParameter.scInSperrAtRükClosed.fbxDoesAlarm.proValue > scParameter.scInSperrAtRükClosed.fbxEnable.proValue THEN
		scParameter.scInSperrAtRükClosed.fbxDoesAlarm.proValue := FALSE;
	END_IF	
	
	fbCheckRükClosed(	(*Inputs*)
						xSafetyIn 			:= xRückIsClosed ,
						xReferenceIn 		:= xOnZu,
						(*Parameter*)
						fbxEnSafetyInput	:= scParameter.scInSperrAtRükClosed.fbxDoesAlarm,
						fbtStartTime 		:= scParameter.scInSperrAtRükClosed.fbtDelayStart,
						fbtRunTime 			:= scParameter.scInSperrAtRükClosed.fbtDelayRun,
						(*Fehler Output*)
						xError 				=> xErrorCloseDI );
	
	(*Klappen Rückmeldung zu*)
	IF scParameter.scInSperrAtRükClosed.fbxEnable.proValue THEN
		xIsClose := xRückIsClosed;
	ELSE
		xIsClose := TON_Zu.Q;
	END_IF		
	
	(* Analog *)
	IF scParameter.scInSperrAtActualPosition.fbxDoesAlarm.proValue > scParameter.scInSperrAtActualPosition.fbxEnable.proValue THEN
		scParameter.scInSperrAtActualPosition.fbxDoesAlarm.proValue := FALSE;
	END_IF
	
	IF scParameter.scInSperrAtActualPosition.fbxDoesAlarm.proValue THEN
		
		xStellwertOutOk := rOnY > 0;		
		
		IF rActualPosition > rOnY + scParameter.scInSperrAtActualPosition.fbrMaxDiff.proValue THEN
			xNoDiffAI	:=	FALSE;
		ELSIF rActualPosition < rOnY - scParameter.scInSperrAtActualPosition.fbrMaxDiff.proValue THEN
			xNoDiffAI	:=	FALSE;
		ELSIF rOnY = 0 THEN
			xNoDiffAI	:=	FALSE;		
		ELSE
			xNoDiffAI	:=	TRUE;
		END_IF
		
		fbCheckValueAI(		(*Inputs*)
							xSafetyIn 			:= xNoDiffAI ,
							xReferenceIn 		:= xStellwertOutOk,
							(*Parameter*)
							fbxEnSafetyInput	:= scParameter.scInSperrAtActualPosition.fbxDoesAlarm,
							fbtStartTime 		:= scParameter.scInSperrAtActualPosition.fbtDelayStart,
							fbtRunTime 			:= scParameter.scInSperrAtActualPosition.fbtDelayRun,
							(*Fehler Output*)
							xError 				=> xErrorDiffAI);
	END_IF
	
	(* EWI *)
	actReport();
ELSE
    (* Off if Disabled or Config Error *)

	xOnZu		:=	FALSE;
	xOnAuf		:=	FALSE;
	xIsOpen		:=  FALSE;
    xIsClose	:=  FALSE;
    rOnY		:=    0.0;
    
    (* Reset Flags *)
    actResetOnDisable();
	IF xConfigError THEN
		(* EWI *)
		actReport();
	END_IF
END_IF;

(* State *)
actState();
(* Modbus State *)
actMbState();
(* InfluxDB *)
actTrendLog();

PROPERTY proHandOn : BOOL
SET
IF proHandOn THEN
    scParameter.scManual.fbuiManualState.proValue := 2;
END_IF;
END_SET
GET
proHandOn := xIsHandOn;
END_GET
END_PROPERTY

PROPERTY proAuto : BOOL
SET
IF proAuto THEN
    scParameter.scManual.fbuiManualState.proValue   :=	0; 
END_IF;
END_SET
GET
proAuto := xIsAuto;
END_GET
END_PROPERTY

PROPERTY proHandOff : BOOL
SET
IF proHandOff THEN
    scParameter.scManual.fbuiManualState.proValue 	:= 	1;
END_IF;
END_SET
GET
proHandOff := xIsHandOff;
END_GET
END_PROPERTY

PROPERTY proHandManualClose : BOOL
SET
IF proHandManualClose THEN
	scParameter.scManual.fbuiSchaltBefehl.proValue := 1;
END_IF
END_SET
GET
proHandManualClose := xShouldClose;
END_GET
END_PROPERTY

PROPERTY proHardWareHandModulAktive : BOOL
GET
proHardWareHandModulAktive := xActuatorHand;
END_GET
END_PROPERTY

PROPERTY proHandManualOpen : BOOL
SET

IF proHandManualOpen THEN
	scParameter.scManual.fbuiSchaltBefehl.proValue	:= 2;
END_IF
END_SET
GET
proHandManualOpen := xShouldOpen;
END_GET
END_PROPERTY

ACTION actConfig:
(* Config Fb *)
fbConfigFile();

(* Base Parameter *)
scParameter.scBase.fbxEnable                					(_usiParaNr :=  1, ItfConfigFb := fbConfigFile);
scParameter.scBase.fbxControllMb            					(_usiParaNr :=  2, ItfConfigFb := fbConfigFile);
scParameter.scBase.fbxInvertiert								(_usiParaNr :=	3, itfConfigFb := fbConfigFile);
scParameter.scBase.fbtSettingTime								(_usiParaNr := 	4, itfConfigFb := fbConfigFile);
                                                    			
(* Fuse Parameter *)                                			
scParameter.scFuse.fbxEnable                					(_usiParaNr :=  5, ItfConfigFb := fbconfigFile);
scParameter.scFuse.fbxInputMb               					(_usiParaNr :=  6, ItfConfigFb := fbconfigFile);
scParameter.scFuse.fbxDoesAlarm             					(_usiParaNr :=  7, ItfConfigFb := fbconfigFile);
                                                    			
(* Stellantrieb Fuse Parameter *)                   			
scParameter.scActuatorFuse.fbxEnable           					(_usiParaNr :=  8, ItfConfigFb := fbconfigFile);
scParameter.scActuatorFuse.fbxInputMb          					(_usiParaNr :=  9, ItfConfigFb := fbconfigFile);
scParameter.scActuatorFuse.fbxDoesAlarm        					(_usiParaNr :=  10, ItfConfigFb := fbconfigFile);
                                                    			
(* Revision Switch Parameter *)                     			
scParameter.scInSperrAtRevisionSwitch.fbxEnable  				(_usiParaNr := 11, ItfConfigFb := fbconfigFile);
scParameter.scInSperrAtRevisionSwitch.fbxInputMb 				(_usiParaNr := 12, ItfConfigFb := fbconfigFile);
                                                    			
(* Ready Input Parameter *)                         			
scParameter.scInSperrAtReady.fbxEnable           				(_usiParaNr := 13, ItfConfigFb := fbconfigFile);
scParameter.scInSperrAtReady.fbxInputMb          				(_usiParaNr := 14, ItfConfigFb := fbconfigFile);
                                                    			
(* Stellantrieb Input Hand *)                       			
scParameter.scInSperrAtHand.fbxEnable            				(_usiParaNr := 15, ItfConfigFb := fbconfigFile);
scParameter.scInSperrAtHand.fbxInputMb           				(_usiParaNr := 16, ItfConfigFb := fbconfigFile);
                                                    			
(* Is closed Input Parameter *)                     			
scParameter.scInSperrAtRükClosed.fbxEnable		 				(_usiParaNr := 17, ItfConfigFb := fbconfigFile);             
scParameter.scInSperrAtRükClosed.fbxInputMb      				(_usiParaNr := 18, ItfConfigFb := fbconfigFile);
scParameter.scInSperrAtRükClosed.fbxDoesAlarm    				(_usiParaNr := 19, ItfConfigFb := fbconfigFile);
scParameter.scInSperrAtRükClosed.fbtDelayStart   				(_usiParaNr := 20, ItfConfigFb := fbconfigFile);
scParameter.scInSperrAtRükClosed.fbtDelayRun     				(_usiParaNr := 21, ItfConfigFb := fbconfigFile);
scParameter.scInSperrAtRükClosed.fbiTypeOfAck					(_usiParaNr := 22, itfConfigFb := fbConfigFile,_MinInit := 0,_MaxInit :=2);
scParameter.scInSperrAtRükClosed.fbiMaxErrorRetryAllowed		(_usiParaNr := 23, itfConfigFb := fbConfigFile);
                                                    	    	
(* Is open Input Parameter *)                       	    	
scParameter.scInSperrAtRükOpen.fbxEnable		 				(_usiParaNr := 24, ItfConfigFb := fbconfigFile);             
scParameter.scInSperrAtRükOpen.fbxInputMb        				(_usiParaNr := 25, ItfConfigFb := fbconfigFile);
scParameter.scInSperrAtRükOpen.fbxDoesAlarm      				(_usiParaNr := 26, ItfConfigFb := fbconfigFile);
scParameter.scInSperrAtRükOpen.fbtDelayStart     				(_usiParaNr := 27, ItfConfigFb := fbconfigFile);
scParameter.scInSperrAtRükOpen.fbtDelayRun       				(_usiParaNr := 28, ItfConfigFb := fbconfigFile);
scParameter.scInSperrAtRükOpen.fbiTypeOfAck						(_usiParaNr := 29, itfConfigFb := fbConfigFile,_MinInit := 0,_MaxInit :=2);
scParameter.scInSperrAtRükOpen.fbiMaxErrorRetryAllowed			(_usiParaNr := 30, itfConfigFb := fbConfigFile);
                                                            	
(* Actual value Input Parameter *)                          	
scParameter.scInSperrAtActualPosition.fbxEnable     			(_usiParaNr := 31, ItfConfigFb := fbconfigFile);
scParameter.scInSperrAtActualPosition.fbxInputMb    			(_usiParaNr := 32, ItfConfigFb := fbconfigFile);
scParameter.scInSperrAtActualPosition.fbxDoesAlarm  			(_usiParaNr := 33, ItfConfigFb := fbconfigFile);
scParameter.scInSperrAtActualPosition.fbrMaxDiff    			(_usiParaNr := 34, ItfConfigFb := fbconfigFile);
scParameter.scInSperrAtActualPosition.fbtDelayStart 			(_usiParaNr := 35, ItfConfigFb := fbconfigFile);
scParameter.scInSperrAtActualPosition.fbtDelayRun   			(_usiParaNr := 36, ItfConfigFb := fbconfigFile);
scParameter.scInSperrAtActualPosition.fbiTypeOfAck				(_usiParaNr := 37, itfConfigFb := fbConfigFile,_MinInit := 0,_MaxInit :=2);
scParameter.scInSperrAtActualPosition.fbiMaxErrorRetryAllowed 	(_usiParaNr := 38, itfConfigFb := fbConfigFile);

(* InfluxDb *)
scParameter.scInfluxDb.fbxEnable            					(_usiParaNr := 39, ItfConfigFb := fbconfigFile);

(* Manual Parameter *)
scParameter.scManual.fbxAlowManualOn         					(_usiParaNr := 40, ItfConfigFb := fbconfigFile); 
scParameter.scManual.fbuiManualState        					(_usiParaNr := 41, ItfConfigFb := fbconfigFile);
scParameter.scManual.fbuiSchaltBefehl          					(_usiParaNr := 42, ItfConfigFb := fbconfigFile);

xConfigError := fbConfigFile.xError;
END_ACTION

PROPERTY proConfigError : BOOL
GET
proConfigError := xConfigError;
END_GET
END_PROPERTY

PROPERTY proValveIcon : UINT
GET
proValveIcon := uiValveIcon;
END_GET
SET
uiValveIcon := proValveIcon;
END_SET
END_PROPERTY

PROPERTY p_scActuatorFuse_fbxEnable : CtaSysConfig.ITF_DATATYPE;
GET
p_scActuatorFuse_fbxEnable := scParameter.scActuatorFuse.fbxEnable;
END_GET
END_PROPERTY

PROPERTY p_scActuatorFuse_fbxInputMb : CtaSysConfig.ITF_DATATYPE;
GET
p_scActuatorFuse_fbxInputMb := scParameter.scActuatorFuse.fbxInputMb;
END_GET
END_PROPERTY

PROPERTY p_scActuatorFuse_fbxDoesAlarm : CtaSysConfig.ITF_DATATYPE;
GET
p_scActuatorFuse_fbxDoesAlarm := scParameter.scActuatorFuse.fbxDoesAlarm;
END_GET
END_PROPERTY

PROPERTY p_scBase_fbxEnable : CtaSysConfig.ITF_DATATYPE;
GET
p_scBase_fbxEnable := scParameter.scBase.fbxEnable;
END_GET
END_PROPERTY

PROPERTY p_scBase_fbxControllMb : CtaSysConfig.ITF_DATATYPE;
GET
p_scBase_fbxControllMb := scParameter.scBase.fbxControllMb;
END_GET
END_PROPERTY

PROPERTY p_scBase_fbxInvertiert : CtaSysConfig.ITF_DATATYPE;
GET
p_scBase_fbxInvertiert := scParameter.scBase.fbxInvertiert;
END_GET
END_PROPERTY

PROPERTY p_scBase_fbtSettingTime : CtaSysConfig.ITF_DATATYPE;
GET
p_scBase_fbtSettingTime := scParameter.scBase.fbtSettingTime;
END_GET
END_PROPERTY

PROPERTY p_scFuse_fbxEnable : CtaSysConfig.ITF_DATATYPE;
GET
p_scFuse_fbxEnable := scParameter.scFuse.fbxEnable;
END_GET
END_PROPERTY

PROPERTY p_scFuse_fbxInputMb : CtaSysConfig.ITF_DATATYPE;
GET
p_scFuse_fbxInputMb := scParameter.scFuse.fbxInputMb;
END_GET
END_PROPERTY

PROPERTY p_scFuse_fbxDoesAlarm : CtaSysConfig.ITF_DATATYPE;
GET
p_scFuse_fbxDoesAlarm := scParameter.scFuse.fbxDoesAlarm;
END_GET
END_PROPERTY

PROPERTY p_scInSperrAtRevisionSwitch_fbxEnable : CtaSysConfig.ITF_DATATYPE;
GET
p_scInSperrAtRevisionSwitch_fbxEnable := scParameter.scInSperrAtRevisionSwitch.fbxEnable;
END_GET
END_PROPERTY

PROPERTY p_scInSperrAtRevisionSwitch_fbxInputMb : CtaSysConfig.ITF_DATATYPE;
GET
p_scInSperrAtRevisionSwitch_fbxInputMb := scParameter.scInSperrAtRevisionSwitch.fbxInputMb;
END_GET
END_PROPERTY

PROPERTY p_scInSperrAtReady_fbxEnable : CtaSysConfig.ITF_DATATYPE;
GET
p_scInSperrAtReady_fbxEnable := scParameter.scInSperrAtReady.fbxEnable;
END_GET
END_PROPERTY

PROPERTY p_scInSperrAtReady_fbxInputMb : CtaSysConfig.ITF_DATATYPE;
GET
p_scInSperrAtReady_fbxInputMb := scParameter.scInSperrAtReady.fbxInputMb;
END_GET
END_PROPERTY

PROPERTY p_scInSperrAtHand_fbxEnable : CtaSysConfig.ITF_DATATYPE;
GET
p_scInSperrAtHand_fbxEnable := scParameter.scInSperrAtHand.fbxEnable;
END_GET
END_PROPERTY

PROPERTY p_scInSperrAtHand_fbxInputMb : CtaSysConfig.ITF_DATATYPE;
GET
p_scInSperrAtHand_fbxInputMb := scParameter.scInSperrAtHand.fbxInputMb;
END_GET
END_PROPERTY

PROPERTY p_scInSperrAtRükClosed_fbxEnable : CtaSysConfig.ITF_DATATYPE;
GET
p_scInSperrAtRükClosed_fbxEnable := scParameter.scInSperrAtRükClosed.fbxEnable;
END_GET
END_PROPERTY

PROPERTY p_scInSperrAtRükClosed_fbxInputMb : CtaSysConfig.ITF_DATATYPE;
GET
p_scInSperrAtRükClosed_fbxInputMb := scParameter.scInSperrAtRükClosed.fbxInputMb;
END_GET
END_PROPERTY

PROPERTY p_scInSperrAtRükClosed_fbxDoesAlarm : CtaSysConfig.ITF_DATATYPE;
GET
p_scInSperrAtRükClosed_fbxDoesAlarm := scParameter.scInSperrAtRükClosed.fbxDoesAlarm;
END_GET
END_PROPERTY

PROPERTY p_scInSperrAtRükClosed_fbtDelayStart : CtaSysConfig.ITF_DATATYPE;
GET
p_scInSperrAtRükClosed_fbtDelayStart := scParameter.scInSperrAtRükClosed.fbtDelayStart;
END_GET
END_PROPERTY

PROPERTY p_scInSperrAtRükClosed_fbtDelayRun : CtaSysConfig.ITF_DATATYPE;
GET
p_scInSperrAtRükClosed_fbtDelayRun := scParameter.scInSperrAtRükClosed.fbtDelayRun;
END_GET
END_PROPERTY

PROPERTY p_scInSperrAtRükClosed_fbiTypeOfAck : CtaSysConfig.ITF_DATATYPE;
GET
p_scInSperrAtRükClosed_fbiTypeOfAck := scParameter.scInSperrAtRükClosed.fbiTypeOfAck;
END_GET
END_PROPERTY

PROPERTY p_scInSperrAtRükClosed_fbiMaxErrorRetryAllowed : CtaSysConfig.ITF_DATATYPE;
GET
p_scInSperrAtRükClosed_fbiMaxErrorRetryAllowed := scParameter.scInSperrAtRükClosed.fbiMaxErrorRetryAllowed;
END_GET
END_PROPERTY

PROPERTY p_scInSperrAtRükOpen_fbxEnable : CtaSysConfig.ITF_DATATYPE;
GET
p_scInSperrAtRükOpen_fbxEnable := scParameter.scInSperrAtRükOpen.fbxEnable;
END_GET
END_PROPERTY

PROPERTY p_scInSperrAtRükOpen_fbxInputMb : CtaSysConfig.ITF_DATATYPE;
GET
p_scInSperrAtRükOpen_fbxInputMb := scParameter.scInSperrAtRükOpen.fbxInputMb;
END_GET
END_PROPERTY

PROPERTY p_scInSperrAtRükOpen_fbxDoesAlarm : CtaSysConfig.ITF_DATATYPE;
GET
p_scInSperrAtRükOpen_fbxDoesAlarm := scParameter.scInSperrAtRükOpen.fbxDoesAlarm;
END_GET
END_PROPERTY

PROPERTY p_scInSperrAtRükOpen_fbtDelayStart : CtaSysConfig.ITF_DATATYPE;
GET
p_scInSperrAtRükOpen_fbtDelayStart := scParameter.scInSperrAtRükOpen.fbtDelayStart;
END_GET
END_PROPERTY

PROPERTY p_scInSperrAtRükOpen_fbtDelayRun : CtaSysConfig.ITF_DATATYPE;
GET
p_scInSperrAtRükOpen_fbtDelayRun := scParameter.scInSperrAtRükOpen.fbtDelayRun;
END_GET
END_PROPERTY

PROPERTY p_scInSperrAtRükOpen_fbiTypeOfAck : CtaSysConfig.ITF_DATATYPE;
GET
p_scInSperrAtRükOpen_fbiTypeOfAck := scParameter.scInSperrAtRükOpen.fbiTypeOfAck;
END_GET
END_PROPERTY

PROPERTY p_scInSperrAtRükOpen_fbiMaxErrorRetryAllowed : CtaSysConfig.ITF_DATATYPE;
GET
p_scInSperrAtRükOpen_fbiMaxErrorRetryAllowed := scParameter.scInSperrAtRükOpen.fbiMaxErrorRetryAllowed;
END_GET
END_PROPERTY

PROPERTY p_scInSperrAtActualPosition_fbxEnable : CtaSysConfig.ITF_DATATYPE;
GET
p_scInSperrAtActualPosition_fbxEnable := scParameter.scInSperrAtActualPosition.fbxEnable;
END_GET
END_PROPERTY

PROPERTY p_scInSperrAtActualPosition_fbxInputMb : CtaSysConfig.ITF_DATATYPE;
GET
p_scInSperrAtActualPosition_fbxInputMb := scParameter.scInSperrAtActualPosition.fbxInputMb;
END_GET
END_PROPERTY

PROPERTY p_scInSperrAtActualPosition_fbxDoesAlarm : CtaSysConfig.ITF_DATATYPE;
GET
p_scInSperrAtActualPosition_fbxDoesAlarm := scParameter.scInSperrAtActualPosition.fbxDoesAlarm;
END_GET
END_PROPERTY

PROPERTY p_scInSperrAtActualPosition_fbrMaxDiff : CtaSysConfig.ITF_DATATYPE;
GET
p_scInSperrAtActualPosition_fbrMaxDiff := scParameter.scInSperrAtActualPosition.fbrMaxDiff;
END_GET
END_PROPERTY

PROPERTY p_scInSperrAtActualPosition_fbtDelayStart : CtaSysConfig.ITF_DATATYPE;
GET
p_scInSperrAtActualPosition_fbtDelayStart := scParameter.scInSperrAtActualPosition.fbtDelayStart;
END_GET
END_PROPERTY

PROPERTY p_scInSperrAtActualPosition_fbtDelayRun : CtaSysConfig.ITF_DATATYPE;
GET
p_scInSperrAtActualPosition_fbtDelayRun := scParameter.scInSperrAtActualPosition.fbtDelayRun;
END_GET
END_PROPERTY

PROPERTY p_scInSperrAtActualPosition_fbiTypeOfAck : CtaSysConfig.ITF_DATATYPE;
GET
p_scInSperrAtActualPosition_fbiTypeOfAck := scParameter.scInSperrAtActualPosition.fbiTypeOfAck;
END_GET
END_PROPERTY

PROPERTY p_scInSperrAtActualPosition_fbiMaxErrorRetryAllowed : CtaSysConfig.ITF_DATATYPE;
GET
p_scInSperrAtActualPosition_fbiMaxErrorRetryAllowed := scParameter.scInSperrAtActualPosition.fbiMaxErrorRetryAllowed;
END_GET
END_PROPERTY

PROPERTY p_scManual_fbxAlowManualOn : CtaSysConfig.ITF_DATATYPE;
GET
p_scManual_fbxAlowManualOn := scParameter.scManual.fbxAlowManualOn;
END_GET
END_PROPERTY

PROPERTY p_scManual_fbuiManualState : CtaSysConfig.ITF_DATATYPE;
GET
p_scManual_fbuiManualState := scParameter.scManual.fbuiManualState;
END_GET
END_PROPERTY

PROPERTY p_scManual_fbuiSchaltBefehl : CtaSysConfig.ITF_DATATYPE;
GET
p_scManual_fbuiSchaltBefehl := scParameter.scManual.fbuiSchaltBefehl;
END_GET
END_PROPERTY

PROPERTY p_scInfluxDb_fbxEnable : CtaSysConfig.ITF_DATATYPE;
GET
p_scInfluxDb_fbxEnable := scParameter.scInfluxDb.fbxEnable;
END_GET
END_PROPERTY

ACTION actMbControll:
IF NOT xModbusTest THEN
    (* Controll Word 0 Digital Controll *)
    (* Release from Modbus *)
    IF scParameter.scBase.fbxControllMb.proValue THEN
        xReleaseFromModBus              := ayMbControllWord[0].0; 
    ELSE
        xReleaseFromModBus              := FALSE;
    END_IF;
    (* Actuator Ready *)
    IF scParameter.scInSperrAtReady.fbxInputMb.proValue THEN
        xInActuatorIsReadyMb               := ayMbControllWord[0].2;
    ELSE
        xInActuatorIsReadyMb               := FALSE;
    END_IF;
    (* Actuator is Open *)
   	IF scParameter.scInSperrAtRükOpen.fbxInputMb.proValue THEN
        xInRükIsOpenMb                  := ayMbControllWord[0].3;
    ELSE
        xInRükIsOpenMb                  := FALSE;
    END_IF; 
    (* Actuator is Closed *)
    IF scParameter.scInSperrAtRükClosed.fbxInputMb.proValue THEN
        xInRükIsClosedMb               := ayMbControllWord[0].4;
    ELSE
        xInRükIsClosedMb               := FALSE;
    END_IF;
    (* Revision Switch *)
    IF scParameter.scInSperrAtRevisionSwitch.fbxInputMb.proValue THEN
        xInActuatorRevisionSwitchOnMb      := ayMbControllWord[0].5;
    ELSE
        xInActuatorRevisionSwitchOnMb      := FALSE;    
    END_IF;
    (* Fuse Ok *)
    IF scParameter.scFuse.fbxInputMb.proValue THEN    
        xInFuseOkMb                     := ayMbControllWord[0].6;
    ELSE
        xInFuseOkMb                     := FALSE;
    END_IF;
    (* Actuator Protection *)
    IF scParameter.scActuatorFuse.fbxInputMb.proValue THEN
        xInActuatorFuseOkMb                := ayMbControllWord[0].7;
    ELSE
        xInActuatorFuseOkMb                := FALSE;
    END_IF;
    (* Actuator Hand *)
    IF scParameter.scInSperrAtHand.fbxInputMb.proValue THEN
        xInActuatorHandMb                  := ayMbControllWord[0].8;
    ELSE
        xInActuatorHandMb                  := FALSE;
    END_IF; 
	(* Actual Position*)
	IF scParameter.scInSperrAtActualPosition.fbxInputMb.proValue THEN
		rInActualPositionMb					:= LIMIT(0,TO_REAL(TO_INT(ayMbControllWord[2]))/10,100);
	ELSE  
		rInActualPositionMb					:= 0; 
	END_IF
ELSE
    xReleaseFromModBus              	:= FALSE;
    xInActuatorIsReadyMb               	:= FALSE;
	xInRükIsOpenMb						:= FALSE;
	xInRükIsClosedMb					:= FALSE;
    xInActuatorRevisionSwitchOnMb      	:= FALSE; 
    xInFuseOkMb                     	:= FALSE;
    xInActuatorFuseOkMb                	:= FALSE;
    xInActuatorHandMb                  	:= FALSE;
	rInActualPositionMb					:= 0;
END_IF;
END_ACTION

ACTION actMbState:
IF NOT xModbusTest THEN
    (* State Word 0 Digital Info*)
    ayMbStateWord[0].00     := xOnAuf;
    ayMbStateWord[0].01     := xOnZu;
    ayMbStateWord[0].02     := xActuatorIsReady;
    ayMbStateWord[0].03     := xRückIsOpen;
    ayMbStateWord[0].04     := xRückIsClosed;
    ayMbStateWord[0].05     := xActuatorRevisionSwitchOn;
    ayMbStateWord[0].06     := xFuseOk;
    ayMbStateWord[0].07     := xActuatorFuseOk;
    ayMbStateWord[0].08     := xIsHand;
    ayMbStateWord[0].09     := xIsAuto;
    ayMbStateWord[0].10     := FALSE;
    ayMbStateWord[0].11     := FALSE;
    ayMbStateWord[0].12     := FALSE;
    ayMbStateWord[0].13     := FALSE;
    ayMbStateWord[0].14     := xIsWarning;
    ayMbStateWord[0].15     := xIsError;
    (* State Word 1 setpoint*)
    ayMbStateWord[1]        := TO_WORD((TO_INT(rOnY * 10)));
    (* State Word 2 actual value*)
    ayMbStateWord[2]        := SEL(scParameter.scInSperrAtActualPosition.fbxEnable.proValue,TO_WORD((TO_INT(rOnY * 10))), TO_WORD((TO_INT(rActualPosition * 10))));
END_IF;
END_ACTION

PROPERTY proModbusTest : BOOL
SET
xModbusTest := proModbusTest;
END_SET
GET
proModbusTest := xModbusTest;
END_GET
END_PROPERTY

PROPERTY proModbusStateWord : REFERENCE TO ARRAY[0..3] OF WORD
GET
proModbusStateWord REF= ayMbStateWord;
END_GET
END_PROPERTY

PROPERTY proModbusControllWord : REFERENCE TO ARRAY[0..3] OF WORD
GET
proModbusControllWord REF= ayMbControllWord;
END_GET
END_PROPERTY

PROPERTY proKlappenStatus : enKlappenStatus
GET
IF scParameter.scManual.fbuiManualState.proValue = 0 OR scParameter.scManual.fbuiManualState.proValue = 2  THEN 
	IF xOnZu THEN // Schliessen
		IF NOT proNotShowDI_RükIsClosed THEN			
			IF NOT xRückIsClosed THEN
				proKlappenStatus := enKlappenStatus.Schliesst;
			ELSE				
				proKlappenStatus := enKlappenStatus.IstZu;
			END_IF			
		ELSE
			IF NOT TON_Zu.Q THEN
				proKlappenStatus := enKlappenStatus.Schliesst;
			ELSE
				proKlappenStatus := enKlappenStatus.IstZu;
			END_IF		
		END_IF	
	ELSIF xOnAuf THEN // Öffnen
		IF NOT proNotShowDI_RükIsOpen THEN			
			IF NOT xRückIsOpen THEN
				proKlappenStatus := enKlappenStatus.Öffnet;
			ELSE				
				proKlappenStatus := enKlappenStatus.IstOffen;
			END_IF			
		ELSE
			IF NOT TON_Auf.Q THEN
				proKlappenStatus := enKlappenStatus.Öffnet;
			ELSE
				proKlappenStatus := enKlappenStatus.IstOffen;
			END_IF		
		END_IF		
	ELSE
		proKlappenStatus := enKlappenStatus.Idle;
	END_IF
ELSIF scParameter.scManual.fbuiManualState.proValue = 1 THEN	
	proKlappenStatus := enKlappenStatus.Gesperrt; // Gesperrt
END_IF
END_GET
END_PROPERTY

PROPERTY proIsError : BOOL
GET
proIsError := xIsError;
END_GET
END_PROPERTY

PROPERTY proIsWarning : BOOL
GET
proIsWarning := xIsWarning;
END_GET
END_PROPERTY

PROPERTY proIsRegulatet : BOOL
GET
proIsRegulatet := xIsRegulatet;
END_GET
END_PROPERTY

PROPERTY proIsEnabled : BOOL
GET
proIsEnabled := xIsEnabled;
END_GET
END_PROPERTY

ACTION actState:
xIsWarning        := _xIsWarning;         
xIsError          := _xIsError;                  
xIsEnabled        := scParameter.scBase.fbxEnable.proValue;
xIsInverted		  := scParameter.scBase.fbxInvertiert.proValue; 
xIsHandOn         := scParameter.scManual.fbuiManualState.proValue = 2;         
xIsHandOff        := scParameter.scManual.fbuiManualState.proValue = 1;          
xIsAuto           := scParameter.scManual.fbuiManualState.proValue = 0 AND NOT xActuatorHand; 
xShouldClose	  := scParameter.scManual.fbuiSchaltBefehl.proValue = 1;	
xShouldOpen		  := scParameter.scManual.fbuiSchaltBefehl.proValue = 2;		 
xIsHand           := xIsHandOn OR xIsHandOff OR xActuatorHand;
END_ACTION

PROPERTY proIsHandOnOrOff : BOOL
GET
proIsHandOnOrOff := xIsHand;
END_GET
END_PROPERTY

PROPERTY proIsReady : BOOL
GET
proIsReady := xActuatorIsReady AND NOT xIsError;
END_GET
END_PROPERTY

PROPERTY proIsOnY : REAL
GET
proIsOnY := rActualPosition;
END_GET
END_PROPERTY

PROPERTY proRevisionSwitchOk : BOOL
GET
proRevisionSwitchOk := xActuatorRevisionSwitchOn;
END_GET
END_PROPERTY

PROPERTY proStateSymbol : STRING
GET
IF xIsError THEN
    proStateSymbol := 'CtaVisSymbols.ImagePool.CtaError';
ELSE    
    IF xIsWarning THEN
        IF scEWI.iWarning = 2 THEN
            proStateSymbol := 'CtaVisSymbols.ImagePool.front_hand_Yellow_Off';
        ELSIF scEWI.iWarning = 3 THEN
            proStateSymbol := 'CtaVisSymbols.ImagePool.front_hand_Yellow';
        ELSE
            proStateSymbol := 'CtaVisSymbols.ImagePool.CtaWarning';
        END_IF;
     ELSE
         proStateSymbol := '';
	 END_IF
END_IF;
END_GET
END_PROPERTY

PROPERTY proAnzError : INT
GET
proAnzError := fbReportManager.proAnzError;
END_GET
END_PROPERTY

PROPERTY proAnzInfo : INT
GET
proAnzInfo := fbReportManager.proAnzInfo;
END_GET
END_PROPERTY

PROPERTY proAnzWarning : INT
GET
proAnzWarning := fbReportManager.proAnzWarning;
END_GET
END_PROPERTY

PROPERTY proITF_REPORTMANAGER : CtaAppReport.ITF_REPORTMANAGER
GET
proITF_REPORTMANAGER := fbReportManager;
END_GET
END_PROPERTY

PROPERTY proIsInverted : BOOL
GET
proIsInverted := xIsInverted;
END_GET
END_PROPERTY

PROPERTY proRükIsClosed : BOOL
GET
proRükIsClosed := xRückIsClosed;
END_GET
END_PROPERTY

PROPERTY proRükIsOpen : BOOL
GET
proRükIsOpen := xRückIsOpen;
END_GET
END_PROPERTY

PROPERTY proOn : BOOL
GET
proOn := xReleaseControllPrio;
END_GET
END_PROPERTY

METHOD metDI_RükIsOpen
VAR_INPUT
    ITF_IN		:	CtaSysIO.ITF_IO;
END_VAR
VAR	
	ITF_DI		:	CtaSysIO.ITF_DI;
END_VAR
IF ITF_IN <> 0 THEN
	ITF_RükIsOpen := ITF_IN;
	IF __QUERYINTERFACE(ITF_RükIsOpen,ITF_DI) THEN
		xInRükIsOpen := ITF_DI.proValue;
	END_IF
ELSE
	xInRükIsOpen := 0;
END_IF
END_METHOD

PROPERTY proGetDI_RükIsOpen : BOOL
GET
proGetDI_RükIsOpen := xInRükIsOpen;
END_GET
END_PROPERTY

PROPERTY proNotShowDI_RükIsOpen : BOOL
GET
proNotShowDI_RükIsOpen := NOT scParameter.scInSperrAtRükOpen.fbxEnable.xValue OR scParameter.scInSperrAtRükOpen.fbxInputMb.xValue;
END_GET
END_PROPERTY

PROPERTY proIsOpen_ITF : CtaSysIO.ITF_IO
GET
proIsOpen_ITF := ITF_RükIsOpen;
END_GET
END_PROPERTY

METHOD metDI_RükIsClosed
VAR_INPUT
    ITF_IN		:	CtaSysIO.ITF_IO;
END_VAR
VAR	
	ITF_DI		:	CtaSysIO.ITF_DI;
END_VAR
IF ITF_IN <> 0 THEN
	ITF_RükIsClosed := ITF_IN;
	IF __QUERYINTERFACE(ITF_RükIsClosed,ITF_DI) THEN
		xInRükIsClosed := ITF_DI.proValue;
	END_IF
ELSE
	xInRükIsClosed := 0;
END_IF
END_METHOD

PROPERTY proGetDI_RükIsClosed : BOOL
GET
proGetDI_RükIsClosed := xInRükIsClosed;
END_GET
END_PROPERTY

PROPERTY proNotShowDI_RükIsClosed : BOOL
GET
proNotShowDI_RükIsClosed := NOT scParameter.scInSperrAtRükClosed.fbxEnable.xValue OR scParameter.scInSperrAtRükClosed.fbxInputMb.xValue;
END_GET
END_PROPERTY

PROPERTY proIsClosed_ITF : CtaSysIO.ITF_IO
GET
proIsClosed_ITF := ITF_RükIsClosed;
END_GET
END_PROPERTY

METHOD metDI_RevisionSwitchOk
VAR_INPUT
    ITF_IN		:	CtaSysIO.ITF_IO;
END_VAR
VAR	
	ITF_DI		:	CtaSysIO.ITF_DI;
END_VAR
IF ITF_IN <> 0 THEN
	ITF_RevisionSwitchOk := ITF_IN;
	IF __QUERYINTERFACE(ITF_RevisionSwitchOk,ITF_DI) THEN
		xInActuatorRevisionSwitchOn := ITF_DI.proValue;
	END_IF
ELSE
	xInActuatorRevisionSwitchOn := 0;
END_IF
END_METHOD

PROPERTY proNotShowDI_RevisionSwitchOk : BOOL
GET
proNotShowDI_RevisionSwitchOk := NOT scParameter.scInSperrAtRevisionSwitch.fbxEnable.xValue OR scParameter.scInSperrAtRevisionSwitch.fbxInputMb.xValue;
END_GET
END_PROPERTY

PROPERTY proGetDI_RevisionSwitchOK : BOOL
GET
proGetDI_RevisionSwitchOK := xInActuatorRevisionSwitchOn;
END_GET
END_PROPERTY

PROPERTY proRevisionSwitch_ITF : CtaSysIO.ITF_IO
GET
proRevisionSwitch_ITF := ITF_RevisionSwitchOk;
END_GET
END_PROPERTY

PROPERTY proGetDI_FuseOK : BOOL
GET
proGetDI_FuseOK := xInFuseOk;
END_GET
END_PROPERTY

METHOD metDI_FuseOK
VAR_INPUT
    ITF_IN		:	CtaSysIO.ITF_IO;
END_VAR
VAR	
	ITF_DI		:	CtaSysIO.ITF_DI;
END_VAR
IF ITF_IN <> 0 THEN
	ITF_FuseOk := ITF_IN;
	IF __QUERYINTERFACE(ITF_FuseOk,ITF_DI) THEN
		xInFuseOk := ITF_DI.proValue;
	END_IF
ELSE
	xInFuseOk := 0;	
END_IF
END_METHOD

PROPERTY proNotShowDI_FuseOk : BOOL
GET
proNotShowDI_FuseOk := NOT scParameter.scFuse.fbxEnable.xValue OR scParameter.scFuse.fbxInputMb.xValue;
END_GET
END_PROPERTY

PROPERTY proFuse_ITF : CtaSysIO.ITF_IO
GET
proFuse_ITF := ITF_FuseOk;
END_GET
END_PROPERTY

METHOD metDI_ActuatorHand
VAR_INPUT
    ITF_IN		:	CtaSysIO.ITF_IO;
END_VAR
VAR	
	ITF_DI		:	CtaSysIO.ITF_DI;
END_VAR
IF ITF_IN <> 0 THEN
	ITF_ActuatorHand := ITF_IN;
	IF __QUERYINTERFACE(ITF_ActuatorHand,ITF_DI) THEN
		xInActuatorHand := ITF_DI.proValue;
	END_IF
ELSE	
	xInActuatorHand := 0;
END_IF
END_METHOD

PROPERTY proNotShowDI_ActuatorHand : BOOL
GET
proNotShowDI_ActuatorHand := NOT scParameter.scInSperrAtHand.fbxEnable.xValue OR scParameter.scInSperrAtHand.fbxInputMb.xValue;
END_GET
END_PROPERTY

PROPERTY proGetDI_ActuatorHand : BOOL
GET
proGetDI_ActuatorHand := xInActuatorHand;
END_GET
END_PROPERTY

PROPERTY proHandModul_ITF : CtaSysIO.ITF_IO
GET
proHandModul_ITF := ITF_ActuatorHand;
END_GET
END_PROPERTY

METHOD metDI_IsReady
VAR_INPUT
    ITF_IN		:	CtaSysIO.ITF_IO;
END_VAR
VAR	
	ITF_DI		:	CtaSysIO.ITF_DI;
END_VAR
IF ITF_IN <> 0 THEN
	ITF_ActuatorIsReady := ITF_IN;
	IF __QUERYINTERFACE(ITF_ActuatorIsReady,ITF_DI) THEN
		xInActuatorIsReady := ITF_DI.proValue;
	END_IF
ELSE
	xInActuatorIsReady := 0;
END_IF
END_METHOD

PROPERTY proNotShowDI_Ready : BOOL
GET
proNotShowDI_Ready := NOT scParameter.scInSperrAtReady.fbxEnable.xValue OR scParameter.scInSperrAtReady.fbxInputMb.xValue;
END_GET
END_PROPERTY

PROPERTY proGetDI_IsReady : BOOL
GET
proGetDI_IsReady := xInActuatorIsReady;
END_GET
END_PROPERTY

PROPERTY proActuatorReady_ITF : CtaSysIO.ITF_IO
GET
proActuatorReady_ITF := ITF_ActuatorIsReady;
END_GET
END_PROPERTY

METHOD metDI_ActuatorFuseOk
VAR_INPUT
    ITF_IN		:	CtaSysIO.ITF_IO;
END_VAR
VAR	
	ITF_DI		:	CtaSysIO.ITF_DI;
END_VAR
IF ITF_IN <> 0 THEN
	ITF_ActuatorFuseOk := ITF_IN;
	IF __QUERYINTERFACE(ITF_ActuatorFuseOk,ITF_DI) THEN
		xInActuatorFuseOk := ITF_DI.proValue;
	END_IF
ELSE	
	xInActuatorFuseOk := 0;
END_IF
END_METHOD

PROPERTY proNotShowDI_ActuatorFuseOk : BOOL
GET
proNotShowDI_ActuatorFuseOk := NOT scParameter.scActuatorFuse.fbxEnable.xValue OR scParameter.scActuatorFuse.fbxInputMb.xValue;
END_GET
END_PROPERTY

PROPERTY proGetDI_ActuatorFuseOk : BOOL
GET
proGetDI_ActuatorFuseOk := xInActuatorFuseOk;
END_GET
END_PROPERTY

PROPERTY proActuatorFuse_ITF : CtaSysIO.ITF_IO
GET
proActuatorFuse_ITF := ITF_ActuatorFuseOk;
END_GET
END_PROPERTY

PROPERTY proActualPosition_ITF : CtaSysIO.ITF_IO
GET
proActualPosition_ITF := ITF_ActualPosition;
END_GET
END_PROPERTY

METHOD metAI_ActualPosition
VAR_INPUT
    ITF_IN		:	CtaSysIO.ITF_IO;
END_VAR
VAR	
	ITF_AI		:	CtaSysIO.ITF_AI;
END_VAR
IF ITF_IN <> 0 THEN
	ITF_ActualPosition := ITF_IN;
	IF __QUERYINTERFACE(ITF_ActualPosition,ITF_AI) THEN
		rInActualPosition := ITF_AI.proValue;
	END_IF
ELSE	
	rInActualPosition := 0;
END_IF
END_METHOD

PROPERTY proNotShowAI_ActualPosition : BOOL
GET
proNotShowAI_ActualPosition := NOT scParameter.scInSperrAtActualPosition.fbxEnable.xValue OR scParameter.scInSperrAtActualPosition.fbxInputMb.xValue;
END_GET
END_PROPERTY

PROPERTY proGetAI_ActualPosition : REAL
GET
proGetAI_ActualPosition := rInActualPosition;
END_GET
END_PROPERTY

PROPERTY proOnY_ITF : CtaSysIO.ITF_IO
GET
proOnY_ITF := ITF_rOnY;
END_GET
END_PROPERTY

METHOD metAO_OnY : REAL
VAR_INPUT
    ITF_IN		:	CtaSysIO.ITF_IO;
END_VAR
VAR	
	ITF_AO		:	CtaSysIO.ITF_AO;
END_VAR
IF ITF_IN <> 0 THEN
	ITF_rOnY := ITF_IN;	
	IF __QUERYINTERFACE(ITF_rOnY,ITF_AO) THEN		
		ITF_AO.proValue := rOnY;
	END_IF	
ELSE
	metAO_OnY := rOnY;
END_IF
END_METHOD

PROPERTY proOnOpen_ITF : CtaSysIO.ITF_IO
GET
proOnOpen_ITF := ITF_xOnAuf;
END_GET
END_PROPERTY

METHOD metDO_xOnAuf : BOOL
VAR_INPUT
    ITF_IN		:	CtaSysIO.ITF_IO;
END_VAR
VAR	
	ITF_DO		:	CtaSysIO.ITF_DO;
END_VAR
IF ITF_IN <> 0 THEN	
	ITF_xOnAuf := ITF_IN;
	IF __QUERYINTERFACE(ITF_xOnAuf,ITF_DO) THEN		
		ITF_DO.proValue := xOnAuf;
	END_IF	
ELSE
	metDO_xOnAuf := xOnAuf;
END_IF
END_METHOD

PROPERTY proOnClose_ITF : CtaSysIO.ITF_IO
GET
proOnClose_ITF := ITF_xOnZu;
END_GET
END_PROPERTY

METHOD metDO_xOnZu : BOOL
VAR_INPUT
    ITF_IN		:	CtaSysIO.ITF_IO;
END_VAR
VAR	
	ITF_DO		:	CtaSysIO.ITF_DO;
END_VAR
IF ITF_IN <> 0 THEN	
	ITF_xOnZu := ITF_IN;
	IF __QUERYINTERFACE(ITF_xOnZu,ITF_DO) THEN		
		ITF_DO.proValue := xOnZu;
	END_IF	
ELSE
	metDO_xOnZu := xOnZu;
END_IF
END_METHOD

PROPERTY proOnY : REAL
GET
proOnY := rOnY;
END_GET
END_PROPERTY

ACTION actPrioOfControll:
(* get Controll request *)
xReleaseControllPrio := SEL(xRelease,xReleaseFromModBus,xRelease);  // xRelease request from Software has prio

(* Get state from Input or ModBus *)

(* Actuall Position from AI *)
// Value Actual Position 0 if not Enabled
rActualPosition						:= SEL(scParameter.scInSperrAtActualPosition.fbxEnable.xValue	,0		,SEL(scParameter.scInSperrAtActualPosition.fbxInputMb.xValue	,rInActualPosition				,rInActualPositionMb			)); 
(* Actuator is Open *)
// Flag RückIsOpen False if not Enabled
xRückIsOpen							:= SEL(scParameter.scInSperrAtRükOpen.fbxEnable.xValue			,FALSE	,SEL(scParameter.scInSperrAtRükOpen.fbxInputMb.xValue			,xInRükIsOpen					,xInRükIsOpenMb					));
(* Actuator is Closed *)
// Flag RückIsClosed False if not Enabled
xRückIsClosed						:= SEL(scParameter.scInSperrAtRükClosed.fbxEnable.xValue		,FALSE	,SEL(scParameter.scInSperrAtRükClosed.fbxInputMb.xValue			,xInRükIsClosed					,xInRükIsClosedMb				));
(* Fuse ok *)
// Flag FuseOk True if not Enabled
xFuseOk								:= SEL(scParameter.scFuse.fbxEnable.xValue					,TRUE	,SEL(scParameter.scFuse.fbxInputMb.xValue					,xInFuseOk						,xInFuseOkMb                	));                     
(* Motor fuse ok *)
// Flag MotorFuseOk True if not Enabled
xActuatorFuseOk						:= SEL(scParameter.scActuatorFuse.fbxEnable.xValue			,TRUE	,SEL(scParameter.scActuatorFuse.fbxInputMb.xValue			,xInActuatorFuseOk				,xInActuatorFuseOkMb           	));
(* Motor is ready *)
// Flag MotorIsReady True if not Enabled
xActuatorIsReady					:= SEL(scParameter.scInSperrAtReady.fbxEnable.xValue			,TRUE	,SEL(scParameter.scInSperrAtReady.fbxInputMb.xValue				,xInActuatorIsReady				,xInActuatorIsReadyMb          	)); 
(* Revision Switch *)
// Flag MotorRevisionSwitchOn True if not Enabled
xActuatorRevisionSwitchOn			:= SEL(scParameter.scInSperrAtRevisionSwitch.fbxEnable.xValue	,TRUE	,SEL(scParameter.scInSperrAtRevisionSwitch.fbxInputMb.xValue	,xInActuatorRevisionSwitchOn	,xInActuatorRevisionSwitchOnMb 	));
xActuatorRevisionSwitchOff			:= NOT xActuatorRevisionSwitchOn;
(* Motor is hand *)
// Flag MotorHand False if not Enabled
xActuatorHand						:= SEL(scParameter.scInSperrAtHand.fbxEnable.xValue				,FALSE	,SEL(scParameter.scInSperrAtHand.fbxInputMb.xValue				,xInActuatorHand				,xInActuatorHandMb             	));
END_ACTION

ACTION actResetOnDisable:
                         
rActualPosition				:= 0	;
xRückIsOpen					:= FALSE;
xRückIsClosed				:= FALSE;
xFuseOk						:= FALSE;    
xActuatorFuseOk				:= FALSE;
xActuatorIsReady			:= FALSE;
xActuatorRevisionSwitchOn	:= FALSE;
xActuatorHand				:= FALSE;
TON_Zu.PT					:=  T#0S;
TON_Zu.IN					:= FALSE;
TON_Zu();
TON_Auf.PT					:=  T#0S;
TON_Auf.IN					:= FALSE;
TON_Auf();
END_ACTION

PROPERTY proOnAuf : BOOL
GET
proOnAuf := xOnAuf;
END_GET
END_PROPERTY

PROPERTY proOnZu : BOOL
GET
proOnZu := xOnZu;
END_GET
END_PROPERTY

PROPERTY proEn : BOOL
SET
xIsEnabled := proEn;
END_SET
GET
proEn := xIsEnabled;
END_GET
END_PROPERTY

PROPERTY proEnSymbol : STRING
GET
IF xIsEnabled THEN
    proEnSymbol := 'CtaVisSymbols.ImagePool.CheckboxChecked_blue';
ELSE    
    proEnSymbol := 'CtaVisSymbols.ImagePool.CheckboxUnchecked_withe'; 
END_IF;
END_GET
END_PROPERTY

ACTION actTrendLog:
(* Stellwert Digital zu*)  
fbTrendxOnZu.ENABLE				:=	scParameter.scBase.fbxEnable.proValue AND
									scParameter.scInfluxDb.fbxEnable.proValue;                                                       		
fbTrendxOnZu.KEY				:=	CONCAT(stObjID,'_xOnZu');	                                  		
fbTrendxOnZu.SET_VALUE			:=	xOnZu;

(* Rückmeldung Digital zu*) 
fbTrendxRückIsClosed.ENABLE		:=	scParameter.scBase.fbxEnable.proValue AND
									scParameter.scInfluxDb.fbxEnable.proValue;                                                      		
fbTrendxRückIsClosed.KEY		:= CONCAT(stObjID,'_xRückIsClosed');                             		
fbTrendxRückIsClosed.SET_VALUE	:=	xRückIsClosed;

(* Stellwert Digital auf*)  
fbTrendxOnAuf.ENABLE			:=	scParameter.scBase.fbxEnable.proValue AND
									scParameter.scInfluxDb.fbxEnable.proValue;                                                      		
fbTrendxOnAuf.KEY				:= 	CONCAT(stObjID,'_xOnAuf');                                    		
fbTrendxOnAuf.SET_VALUE			:=	xOnAuf;

(* Rückmeldung Digital auf*) 
fbTrendxRückIsOpen.ENABLE		:=	scParameter.scBase.fbxEnable.proValue AND
									scParameter.scInfluxDb.fbxEnable.proValue;                                                     	
fbTrendxRückIsOpen.KEY			:=	CONCAT(stObjID,'_xRückIsOpen');                               	
fbTrendxRückIsOpen.SET_VALUE 	:= 	xRückIsOpen	;

(* Stellwert Analog*)  
fbTrendrOnY.ENABLE				:=	scParameter.scBase.fbxEnable.proValue AND
									scParameter.scInfluxDb.fbxEnable.proValue;                                                          	
fbTrendrOnY.KEY					:= 	CONCAT(stObjID,'_rOnY');                                      	
fbTrendrOnY.SET_VALUE			:=	rOnY ;

(* Istwert Analog*) 
fbTrendrIsOnY.ENABLE			:=	scParameter.scBase.fbxEnable.proValue AND
									scParameter.scInfluxDb.fbxEnable.proValue;                                                             	
fbTrendrIsOnY.KEY				:= 	CONCAT(stObjID,'_rIsOnY');                                    	
fbTrendrIsOnY.SET_VALUE			:=	proIsOnY;

(* Fehler*)
fbTrendxError.ENABLE			:=	scParameter.scBase.fbxEnable.proValue AND
									scParameter.scInfluxDb.fbxEnable.proValue;                                                                          	
fbTrendxError.KEY				:= 	CONCAT(stObjID,'_xError');                                    	
fbTrendxError.SET_VALUE			:=	xIsError;
END_ACTION

ACTION actReport:
(* EWI Manager *)
fbReportManager(	stErrorInitReportTextListIn		:=	ADR(GlobalKonstant.stReportTextListError),
					stWarningInitReportTextListIn	:=	ADR(GlobalKonstant.stReportTextListWarning),
					stInfoInitReportTextListIn		:=	ADR(GlobalKonstant.stReportTextListInfo),
					scReportNr						:=	scEWI);
(* Errors *)                        
		(* Stellwert Rückmeldung *)
		ayErrorReporter[1].proPrio	:= 3;
		ayErrorReporter[1].metReport(     		xSetReportIn					:= xErrorDiffAI AND scParameter.scInSperrAtActualPosition.fbxDoesAlarm.proValue AND scParameter.scInSperrAtActualPosition.fbxEnable.proValue,
												iReportID						:= 1,
												enReportTypeIn					:= CtaAppReport.enReportType.Error,  
												enReportAcknowledgeTypeIn   	:= scParameter.scInSperrAtActualPosition.fbiTypeOfAck.proValue,
												tDelay							:= T#0S, 
												ITF_BMK_IN						:= THIS^,			              
												pstReportTextListIn				:= ADR(GlobalKonstant.stReportTextListError),
												stOptionalReportText		    := '',   
												iRetryTilReportLock 		    := scParameter.scInSperrAtActualPosition.fbiMaxErrorRetryAllowed.proValue, 
												xResetCount         		    := FALSE,  
												tReset						    := T#24H); 		

		(* Stellventil keine rückmeldung Zu *)
		ayErrorReporter[2].proPrio	:= 3;    
        ayErrorReporter[2].metReport(     		xSetReportIn					:= xErrorCloseDI AND scParameter.scInSperrAtRükClosed.fbxDoesAlarm.proValue AND scParameter.scInSperrAtRükClosed.fbxEnable.proValue,
												iReportID						:= 2,
												enReportTypeIn					:= CtaAppReport.enReportType.Error,  
												enReportAcknowledgeTypeIn   	:= scParameter.scInSperrAtRükClosed.fbiTypeOfAck.proValue,
												tDelay							:= T#0S, 
												ITF_BMK_IN						:= THIS^,			              
												pstReportTextListIn				:= ADR(GlobalKonstant.stReportTextListError),
												stOptionalReportText		    := '',   
												iRetryTilReportLock 		    := scParameter.scInSperrAtRükClosed.fbiMaxErrorRetryAllowed.proValue, 
												xResetCount         		    := FALSE,  
												tReset						    := T#24H); 	  
		(* Stellventil keine rückmeldung Auf *) 
		ayErrorReporter[3].proPrio	:= 3;
		ayErrorReporter[3].metReport(     		xSetReportIn					:= xErrorOpenDI AND scParameter.scInSperrAtRükOpen.fbxDoesAlarm.proValue AND scParameter.scInSperrAtRükOpen.fbxEnable.proValue,
												iReportID						:= 3,
												enReportTypeIn					:= CtaAppReport.enReportType.Error,  
												enReportAcknowledgeTypeIn   	:= scParameter.scInSperrAtRükOpen.fbiTypeOfAck.proValue,
												tDelay							:= T#1S, 
												ITF_BMK_IN						:= THIS^,			              
												pstReportTextListIn				:= ADR(GlobalKonstant.stReportTextListError),
												stOptionalReportText		    := '',   
												iRetryTilReportLock 		    := scParameter.scInSperrAtRükOpen.fbiMaxErrorRetryAllowed.proValue, 
												xResetCount         		    := FALSE,  
												tReset						    := T#24H);
		                   
		(* Error Fuse *)
		ayErrorReporter[4].proPrio	:= 2;    
		ayErrorReporter[4].metReport(     		xSetReportIn					:= NOT xFuseOk AND scParameter.scFuse.fbxDoesAlarm.proValue AND scParameter.scFuse.fbxEnable.proValue,
												iReportID						:= 4,
												enReportTypeIn					:= CtaAppReport.enReportType.Error,  
												enReportAcknowledgeTypeIn   	:= CtaAppReport.enReportacknowledgeType.Auto,
												tDelay							:= T#1S, 
												ITF_BMK_IN						:= THIS^,			              
												pstReportTextListIn				:= ADR(GlobalKonstant.stReportTextListError),
												stOptionalReportText		    := '',   
												iRetryTilReportLock 		    := 0, 
												xResetCount         		    := FALSE,  
												tReset						    := T#24H);
                                                
		(* Error Actuator Fuse *) 
		ayErrorReporter[5].proPrio	:= 2;   
		ayErrorReporter[5].metReport(     		xSetReportIn					:= NOT xActuatorFuseOk AND scParameter.scActuatorFuse.fbxDoesAlarm.proValue AND scParameter.scActuatorFuse.fbxEnable.proValue,
												iReportID						:= 5,
												enReportTypeIn					:= CtaAppReport.enReportType.Error,  
												enReportAcknowledgeTypeIn   	:= CtaAppReport.enReportacknowledgeType.Auto,
												tDelay							:= T#1S, 
												ITF_BMK_IN						:= THIS^,			              
												pstReportTextListIn				:= ADR(GlobalKonstant.stReportTextListError),
												stOptionalReportText		    := '',   
												iRetryTilReportLock 		    := 0, 
												xResetCount         		    := FALSE,  
												tReset						    := T#24H);                                                

		(* Config Error *)
		ayErrorReporter[6].proPrio	:= 1;    
		ayErrorReporter[6].metReport(     		xSetReportIn					:= xConfigError,
												iReportID						:= 6,
												enReportTypeIn					:= CtaAppReport.enReportType.Error,  
												enReportAcknowledgeTypeIn   	:= CtaAppReport.enReportacknowledgeType.Quit,
												tDelay							:= T#1S, 
												ITF_BMK_IN						:= THIS^,			              
												pstReportTextListIn				:= ADR(GlobalKonstant.stReportTextListError),
												stOptionalReportText		    := '',   
												iRetryTilReportLock 		    := 0, 
												xResetCount         		    := FALSE,  
												tReset						    := T#24H);                                           
(* Warnungen *)
		(* Warnung Revisionsschalter Aus *)
		ayWarningReporter[1].proPrio	:= 1;
		ayWarningReporter[1].proHandLokal :=   	xActuatorRevisionSwitchOff; 
		ayWarningReporter[1].metReport(			xSetReportIn					:= xActuatorRevisionSwitchOff,
												iReportID						:= 1,
												enReportTypeIn					:= CtaAppReport.enReportType.Warning,  
												enReportAcknowledgeTypeIn   	:= CtaAppReport.enReportAcknowledgeType.Auto,
												tDelay							:= T#0S, 
												ITF_BMK_IN						:= THIS^,			              
												pstReportTextListIn				:= ADR(GlobalKonstant.stReportTextListWarning),
												stOptionalReportText		    := '',   
												iRetryTilReportLock 		    := 0, 
												xResetCount         		    := FALSE,  
												tReset						    := T#0S);     

		(* Warnung Hand Aus *)
		ayWarningReporter[2].proPrio	:= 3;        
		ayWarningReporter[2].proHandLokal :=    xIsHandOff; 
		ayWarningReporter[2].metReport(			xSetReportIn					:= xIsHandOff,
												iReportID						:= 2,
												enReportTypeIn					:= CtaAppReport.enReportType.Warning,  
												enReportAcknowledgeTypeIn   	:= CtaAppReport.enReportAcknowledgeType.Auto,
												tDelay							:= T#0S, 
												ITF_BMK_IN						:= THIS^,			              
												pstReportTextListIn				:= ADR(GlobalKonstant.stReportTextListWarning),
												stOptionalReportText		    := '',   
												iRetryTilReportLock 		    := 0, 
												xResetCount         		    := FALSE,  
												tReset						    := T#0S);                                  
                                
        (* Warnung Hand Ein *)
		ayWarningReporter[3].proPrio	:= 3;    
		ayWarningReporter[3].proHandLokal :=    xIsHandOn;
		ayWarningReporter[3].metReport(			xSetReportIn					:= xIsHandOn,
												iReportID						:= 3,
												enReportTypeIn					:= CtaAppReport.enReportType.Warning,  
												enReportAcknowledgeTypeIn   	:= CtaAppReport.enReportAcknowledgeType.Auto,
												tDelay							:= T#0S, 
												ITF_BMK_IN						:= THIS^,			              
												pstReportTextListIn				:= ADR(GlobalKonstant.stReportTextListWarning),
												stOptionalReportText		    := '',   
												iRetryTilReportLock 		    := 0, 
												xResetCount         		    := FALSE,  
												tReset						    := T#0S);   
 
        (* Warnung Handmodul Actuator *)
		ayWarningReporter[4].proPrio	:= 4;    
		ayWarningReporter[4].proHandLokal :=    xActuatorHand;
		ayWarningReporter[4].metReport(			xSetReportIn					:= xActuatorHand,
												iReportID						:= 4,
												enReportTypeIn					:= CtaAppReport.enReportType.Warning,  
												enReportAcknowledgeTypeIn   	:= CtaAppReport.enReportAcknowledgeType.Auto,
												tDelay							:= T#0S, 
												ITF_BMK_IN						:= THIS^,			              
												pstReportTextListIn				:= ADR(GlobalKonstant.stReportTextListWarning),
												stOptionalReportText		    := '',   
												iRetryTilReportLock 		    := 0, 
												xResetCount         		    := FALSE,  
												tReset						    := T#0S);                                                   
(* Sync Reports *)                                         
FOR difor := LOWER_BOUND(ayErrorReporter,1) TO UPPER_BOUND(ayErrorReporter,1) DO
	fbReportManager.metSyncReporter(ayErrorReporter[difor]);	
END_FOR;
FOR difor := LOWER_BOUND(ayWarningReporter,1) TO UPPER_BOUND(ayWarningReporter,1) DO
	fbReportManager.metSyncReporter(ayWarningReporter[difor]);	
END_FOR;
                                                                             
_xIsError   := scEWI.iError <> 0;
_xIsWarning := scEWI.iWarning <> 0;
END_ACTION

{attribute 'monitoring' := 'variable'}
PROPERTY proAcknowlege : BOOL
GET
proAcknowlege :=NOT proIsError;
END_GET
END_PROPERTY

{attribute 'monitoring' := 'variable'}
PROPERTY proAvailable : BOOL
GET
proAvailable := proIsReady;
END_GET
END_PROPERTY

